C03632=1082.087,-21.908,442.728,174.022,19.619,153.310
C03633=1082.093,-21.658,442.716,174.024,19.621,153.310
C03634=1082.099,-21.409,442.702,174.025,19.623,153.310
C03635=1082.104,-21.158,442.689,174.026,19.625,153.311
C03636=1082.110,-20.909,442.676,174.028,19.627,153.311
C03637=1082.116,-20.659,442.663,174.030,19.629,153.311
C03638=1082.122,-20.410,442.650,174.031,19.631,153.311
C03639=1082.128,-20.160,442.636,174.032,19.633,153.311
C03640=1082.134,-19.910,442.624,174.034,19.635,153.311
C03641=1082.140,-19.661,442.610,174.035,19.637,153.311
C03642=1082.146,-19.411,442.598,174.037,19.639,153.311
C03643=1082.152,-19.162,442.585,174.039,19.641,153.312
C03644=1082.157,-18.912,442.571,174.040,19.643,153.312
C03645=1082.164,-18.663,442.558,174.041,19.645,153.312
C03646=1082.170,-18.413,442.545,174.042,19.647,153.312
C03647=1082.176,-18.163,442.532,174.045,19.649,153.312
C03648=1082.181,-17.914,442.518,174.046,19.651,153.312
C03649=1082.187,-17.664,442.506,174.047,19.653,153.312
C03650=1082.194,-17.391,442.491,174.048,19.655,153.313
C03651=1082.200,-17.116,442.477,174.050,19.658,153.313
C03652=1082.206,-16.843,442.462,174.052,19.660,153.313
C03653=1082.213,-16.568,442.448,174.054,19.662,153.313
C03654=1082.220,-16.319,442.435,174.055,19.664,153.313
C03655=1082.225,-16.069,442.421,174.056,19.666,153.313
C03656=1082.231,-15.819,442.408,174.058,19.668,153.313
C03657=1082.237,-15.570,442.395,174.059,19.670,153.314
C03658=1082.243,-15.321,442.382,174.061,19.672,153.314
C03659=1082.249,-15.071,442.369,174.063,19.674,153.314
C03660=1082.255,-14.821,442.355,174.064,19.676,153.314
C03661=1082.260,-14.572,442.341,174.065,19.678,153.314
C03662=1082.266,-14.322,442.329,174.066,19.680,153.314
C03663=1082.272,-14.073,442.316,174.068,19.682,153.314
C03664=1082.278,-13.823,442.302,174.070,19.684,153.314
C03665=1082.284,-13.574,442.288,174.071,19.686,153.315
C03666=1082.289,-13.324,442.275,174.072,19.688,153.315
C03667=1082.295,-13.074,442.262,174.074,19.690,153.315
C03668=1082.301,-12.825,442.248,174.076,19.692,153.315
C03669=1082.307,-12.576,442.235,174.077,19.694,153.315
C03670=1082.312,-12.325,442.222,174.078,19.696,153.315
C03671=1082.319,-12.076,442.208,174.079,19.698,153.316
C03672=1082.324,-11.827,442.195,174.082,19.700,153.316
C03673=1082.330,-11.577,442.181,174.083,19.702,153.316
C03674=1082.336,-11.328,442.167,174.084,19.704,153.316
C03675=1082.342,-11.078,442.155,174.085,19.706,153.316
C03676=1082.348,-10.828,442.141,174.087,19.708,153.316
C03677=1082.354,-10.578,442.127,174.089,19.711,153.316
C03678=1082.360,-10.329,442.114,174.090,19.713,153.317
C03679=1082.366,-10.079,442.100,174.091,19.714,153.317
C03680=1082.372,-9.830,442.087,174.093,19.716,153.317
C03681=1082.377,-9.580,442.074,174.095,19.719,153.317
C03682=1082.383,-9.331,442.061,174.096,19.721,153.317
C03683=1082.389,-9.081,442.047,174.097,19.723,153.317
C03684=1082.395,-8.832,442.033,174.099,19.725,153.318
C03685=1082.400,-8.582,442.020,174.100,19.727,153.318
C03686=1082.407,-8.333,442.006,174.102,19.729,153.318
C03687=1082.413,-8.083,441.992,174.103,19.731,153.318
C03688=1082.418,-7.833,441.978,174.105,19.733,153.318
C03689=1082.424,-7.584,441.965,174.106,19.735,153.318
C03690=1082.430,-7.334,441.952,174.108,19.738,153.318
C03691=1082.436,-7.084,441.939,174.109,19.740,153.319
C03692=1082.441,-6.835,441.925,174.110,19.742,153.319
C03693=1082.447,-6.586,441.911,174.112,19.743,153.319
C03694=1082.454,-6.335,441.897,174.113,19.745,153.319
C03695=1082.460,-6.086,441.884,174.115,19.748,153.319
C03696=1082.465,-5.837,441.870,174.117,19.750,153.319
C03697=1082.471,-5.587,441.857,174.118,19.752,153.319
C03698=1082.477,-5.338,441.843,174.119,19.754,153.320
C03699=1082.483,-5.088,441.830,174.121,19.756,153.320
C03700=1082.489,-4.839,441.816,174.123,19.758,153.320
C03701=1082.495,-4.589,441.802,174.124,19.760,153.320
C03702=1082.501,-4.339,441.788,174.125,19.762,153.320
C03703=1082.506,-4.090,441.774,174.127,19.764,153.320
C03704=1082.513,-3.840,441.761,174.128,19.766,153.320
C03705=1082.518,-3.591,441.747,174.130,19.768,153.321
C03706=1082.525,-3.341,441.734,174.131,19.770,153.321
C03707=1082.530,-3.091,441.720,174.132,19.772,153.321
C03708=1082.536,-2.842,441.706,174.134,19.775,153.321
C03709=1082.541,-2.592,441.692,174.136,19.776,153.321
C03710=1082.548,-2.343,441.679,174.137,19.778,153.321
C03711=1082.553,-2.094,441.664,174.138,19.780,153.321
C03712=1082.559,-1.844,441.650,174.140,19.783,153.322
C03713=1082.565,-1.594,441.636,174.142,19.785,153.322
C03714=1082.571,-1.319,441.621,174.143,19.787,153.322
C03715=1082.577,-1.043,441.605,174.145,19.790,153.322
C03716=1082.584,-0.768,441.591,174.146,19.792,153.322
C03717=1082.590,-0.492,441.575,174.148,19.794,153.322
C03718=1082.596,-0.243,441.561,174.149,19.796,153.323
C03719=1082.602,0.007,441.548,174.151,19.798,153.323
C03720=1082.607,0.256,441.534,174.153,19.801,153.323
C03721=1082.613,0.507,441.520,174.154,19.803,153.323
C03722=1082.619,0.756,441.506,174.155,19.805,153.323
C03723=1082.625,1.005,441.492,174.156,19.807,153.323
C03724=1082.631,1.255,441.478,174.158,19.809,153.324
C03725=1082.636,1.504,441.464,174.160,19.811,153.324
C03726=1082.642,1.754,441.450,174.161,19.813,153.324
C03727=1082.648,2.004,441.436,174.162,19.815,153.324
C03728=1082.653,2.253,441.421,174.164,19.818,153.324
C03729=1082.660,2.502,441.408,174.166,19.820,153.324
C03730=1082.665,2.752,441.394,174.167,19.821,153.324
C03731=1082.671,3.002,441.380,174.168,19.823,153.325
C03732=1082.677,3.252,441.366,174.170,19.826,153.325
C03733=1082.682,3.501,441.351,174.172,19.828,153.325
C03734=1082.688,3.750,441.338,174.173,19.830,153.325
C03735=1082.694,4.000,441.323,174.174,19.832,153.325
C03736=1082.701,4.249,441.309,174.176,19.834,153.325
C03737=1082.706,4.499,441.296,174.178,19.836,153.326
C03738=1082.711,4.748,441.282,174.179,19.838,153.326
C03739=1082.718,4.999,441.267,174.180,19.840,153.326
C03740=1082.723,5.247,441.253,174.182,19.843,153.326
C03741=1082.729,5.497,441.239,174.183,19.845,153.326
C03742=1082.734,5.747,441.225,174.185,19.847,153.326
C03743=1082.741,5.996,441.210,174.186,19.849,153.327
C03744=1082.747,6.246,441.197,174.188,19.851,153.327
C03745=1082.752,6.495,441.183,174.189,19.853,153.327
C03746=1082.759,6.745,441.168,174.190,19.855,153.327
C03747=1082.764,6.994,441.154,174.192,19.857,153.327
C03748=1082.770,7.244,441.140,174.194,19.859,153.327
C03749=1082.776,7.494,441.125,174.195,19.861,153.327
C03750=1082.782,7.743,441.112,174.197,19.863,153.328
C03751=1082.787,7.993,441.098,174.199,19.866,153.328
C03752=1082.793,8.242,441.083,174.200,19.868,153.328
C03753=1082.799,8.492,441.069,174.201,19.870,153.328
C03754=1082.805,8.741,441.055,174.202,19.872,153.328
C03755=1082.811,8.991,441.041,174.205,19.874,153.328
C03756=1082.817,9.240,441.026,174.206,19.876,153.329
C03757=1082.823,9.489,441.012,174.207,19.878,153.329
C03758=1082.829,9.740,440.998,174.208,19.880,153.329
C03759=1082.835,9.989,440.983,174.210,19.883,153.329
C03760=1082.840,10.238,440.970,174.212,19.884,153.329
C03761=1082.846,10.488,440.955,174.213,19.886,153.329
C03762=1082.852,10.737,440.941,174.214,19.888,153.330
C03763=1082.858,10.986,440.926,174.217,19.891,153.330
C03764=1082.864,11.237,440.912,174.218,19.893,153.330
C03765=1082.870,11.486,440.897,174.219,19.895,153.330
C03766=1082.876,11.736,440.883,174.221,19.897,153.330
C03767=1082.881,11.985,440.869,174.222,19.899,153.330
C03768=1082.887,12.234,440.855,174.224,19.902,153.330
C03769=1082.893,12.484,440.840,174.225,19.904,153.331
C03770=1082.899,12.734,440.826,174.227,19.906,153.331
C03771=1082.905,12.983,440.811,174.228,19.907,153.331
C03772=1082.911,13.233,440.797,174.230,19.909,153.331
C03773=1082.917,13.482,440.783,174.231,19.911,153.331
C03774=1082.924,13.731,440.768,174.233,19.914,153.331
C03775=1082.929,13.981,440.754,174.234,19.916,153.332
C03776=1082.935,14.230,440.739,174.236,19.918,153.332
C03777=1082.941,14.480,440.725,174.238,19.920,153.332
C03778=1082.947,14.757,440.709,174.239,19.922,153.332
C03779=1082.954,15.035,440.693,174.241,19.925,153.332
C03780=1082.960,15.313,440.677,174.242,19.927,153.332
C03781=1082.967,15.590,440.661,174.244,19.930,153.333
C03782=1082.972,15.840,440.646,174.245,19.932,153.333
C03783=1082.978,16.089,440.631,174.247,19.934,153.333
C03784=1082.984,16.339,440.616,174.249,19.936,153.333
C03785=1082.990,16.588,440.602,174.250,19.938,153.333
C03786=1082.995,16.837,440.588,174.252,19.940,153.333
C03787=1083.002,17.087,440.573,174.253,19.942,153.333
C03788=1083.006,17.337,440.558,174.255,19.944,153.334
C03789=1083.013,17.587,440.543,174.256,19.946,153.334
C03790=1083.019,17.836,440.529,174.257,19.948,153.334
C03791=1083.025,18.086,440.515,174.260,19.951,153.334
C03792=1083.030,18.335,440.500,174.261,19.953,153.334
C03793=1083.035,18.584,440.485,174.262,19.955,153.334
C03794=1083.042,18.834,440.471,174.263,19.957,153.335
C03795=1083.047,19.083,440.456,174.265,19.959,153.335
C03796=1083.054,19.333,440.441,174.267,19.961,153.335
C03797=1083.059,19.582,440.426,174.268,19.963,153.335
C03798=1083.065,19.833,440.412,174.270,19.966,153.335
C03799=1083.071,20.081,440.397,174.271,19.968,153.335
C03800=1083.077,20.331,440.382,174.273,19.970,153.336
C03801=1083.083,20.580,440.368,174.275,19.972,153.336
C03802=1083.088,20.831,440.353,174.276,19.974,153.336
C03803=1083.094,21.080,440.338,174.277,19.976,153.336
C03804=1083.100,21.329,440.324,174.278,19.978,153.336
C03805=1083.105,21.579,440.308,174.281,19.981,153.336
C03806=1083.111,21.828,440.293,174.282,19.983,153.337
C03807=1083.117,22.078,440.279,174.283,19.985,153.337
C03808=1083.123,22.327,440.265,174.285,19.987,153.337
C03809=1083.129,22.577,440.249,174.286,19.989,153.337
C03810=1083.134,22.826,440.235,174.288,19.991,153.337
C03811=1083.141,23.075,440.220,174.290,19.993,153.337
C03812=1083.146,23.325,440.204,174.291,19.995,153.337
C03813=1083.152,23.574,440.189,174.293,19.997,153.338
C03814=1083.158,23.824,440.176,174.294,19.999,153.338
C03815=1083.163,24.074,440.160,174.296,20.002,153.338
C03816=1083.169,24.323,440.145,174.297,20.004,153.338
C03817=1083.175,24.573,440.130,174.298,20.006,153.338
C03818=1083.181,24.822,440.115,174.301,20.008,153.338
C03819=1083.187,25.071,440.100,174.302,20.010,153.339
C03820=1083.192,25.321,440.085,174.303,20.012,153.339
C03821=1083.198,25.570,440.070,174.305,20.015,153.339
C03822=1083.204,25.819,440.056,174.306,20.017,153.339
C03823=1083.210,26.069,440.040,174.308,20.019,153.339
C03824=1083.216,26.319,440.025,174.310,20.021,153.339
C03825=1083.222,26.568,440.011,174.311,20.023,153.340
C03826=1083.227,26.818,439.996,174.312,20.025,153.340
C03827=1083.233,27.067,439.981,174.315,20.028,153.340
C03828=1083.239,27.317,439.966,174.316,20.030,153.340
C03829=1083.244,27.566,439.951,174.317,20.031,153.340
C03830=1083.251,27.816,439.936,174.319,20.033,153.340
C03831=1083.256,28.065,439.921,174.321,20.036,153.340
C03832=1083.262,28.315,439.906,174.322,20.038,153.341
C03833=1083.268,28.565,439.891,174.323,20.040,153.341
C03834=1083.274,28.813,439.875,174.325,20.042,153.341
C03835=1083.280,29.063,439.860,174.327,20.044,153.341
C03836=1083.285,29.312,439.845,174.328,20.046,153.341
C03837=1083.291,29.562,439.830,174.330,20.049,153.341
C03838=1083.297,29.811,439.815,174.331,20.051,153.342
C03839=1083.303,30.061,439.799,174.332,20.053,153.342
C03840=1083.308,30.310,439.785,174.335,20.055,153.342
C03841=1083.314,30.560,439.769,174.336,20.057,153.342
C03842=1083.321,30.839,439.753,174.338,20.060,153.342
C03843=1083.327,31.118,439.735,174.339,20.062,153.342
C03844=1083.333,31.397,439.719,174.341,20.065,153.343
C03845=1083.340,31.676,439.701,174.342,20.067,153.343
C03846=1083.345,31.925,439.687,174.344,20.069,153.343
C03847=1083.351,32.175,439.670,174.346,20.071,153.343
C03848=1083.357,32.424,439.656,174.347,20.073,153.343
C03849=1083.363,32.674,439.640,174.349,20.076,153.343
C03850=1083.368,32.924,439.625,174.351,20.077,153.343
C03851=1083.374,33.173,439.610,174.352,20.079,153.344
C03852=1083.380,33.422,439.595,174.354,20.082,153.344
C03853=1083.386,33.672,439.580,174.355,20.084,153.344
C03854=1083.392,33.921,439.564,174.357,20.086,153.344
C03855=1083.397,34.171,439.548,174.359,20.088,153.344
C03856=1083.403,34.420,439.534,174.360,20.090,153.344
C03857=1083.409,34.670,439.518,174.361,20.092,153.345
C03858=1083.415,34.919,439.502,174.363,20.095,153.345
C03859=1083.420,35.168,439.487,174.365,20.097,153.345
C03860=1083.426,35.418,439.472,174.366,20.099,153.345
C03861=1083.432,35.668,439.457,174.368,20.101,153.345
C03862=1083.437,35.917,439.442,174.369,20.103,153.345
C03863=1083.444,36.166,439.426,174.371,20.105,153.345
C03864=1083.450,36.416,439.410,174.373,20.107,153.346
C03865=1083.455,36.665,439.395,174.374,20.109,153.346
C03866=1083.462,36.914,439.380,174.375,20.111,153.346
C03867=1083.467,37.164,439.364,174.377,20.113,153.346
C03868=1083.472,37.413,439.349,174.379,20.115,153.346
C03869=1083.479,37.662,439.333,174.380,20.117,153.346
C03870=1083.485,37.912,439.318,174.382,20.120,153.347
C03871=1083.490,38.162,439.302,174.383,20.122,153.347
C03872=1083.496,38.411,439.288,174.385,20.124,153.347
C03873=1083.502,38.661,439.271,174.387,20.126,153.347
C03874=1083.508,38.911,439.256,174.388,20.128,153.347
C03875=1083.513,39.159,439.240,174.390,20.131,153.347
C03876=1083.519,39.409,439.224,174.392,20.132,153.347
C03877=1083.525,39.659,439.209,174.393,20.134,153.348
C03878=1083.530,39.908,439.194,174.395,20.137,153.348
C03879=1083.536,40.158,439.178,174.396,20.139,153.348
C03880=1083.542,40.408,439.162,174.398,20.141,153.348
C03881=1083.547,40.656,439.147,174.400,20.143,153.348
C03882=1083.553,40.906,439.132,174.401,20.145,153.348
C03883=1083.559,41.155,439.115,174.402,20.147,153.349
C03884=1083.564,41.404,439.100,174.404,20.150,153.349
C03885=1083.570,41.654,439.084,174.406,20.152,153.349
C03886=1083.576,41.904,439.068,174.407,20.154,153.349
C03887=1083.582,42.153,439.053,174.409,20.156,153.349
C03888=1083.588,42.402,439.038,174.410,20.158,153.349
C03889=1083.593,42.652,439.022,174.412,20.161,153.350
C03890=1083.599,42.901,439.006,174.414,20.162,153.350
C03891=1083.605,43.151,438.990,174.415,20.164,153.350
C03892=1083.610,43.400,438.974,174.417,20.167,153.350
C03893=1083.617,43.650,438.959,174.419,20.169,153.350
C03894=1083.623,43.899,438.943,174.420,20.171,153.350
C03895=1083.628,44.149,438.928,174.422,20.173,153.350
C03896=1083.634,44.398,438.912,174.423,20.175,153.351
C03897=1083.639,44.648,438.896,174.424,20.177,153.351
C03898=1083.645,44.897,438.880,174.427,20.180,153.351
C03899=1083.650,45.146,438.865,174.428,20.182,153.351
C03900=1083.656,45.396,438.848,174.430,20.184,153.351
C03901=1083.662,45.645,438.832,174.431,20.186,153.351
C03902=1083.668,45.895,438.817,174.433,20.188,153.352
C03903=1083.673,46.144,438.801,174.435,20.190,153.352
C03904=1083.678,46.394,438.785,174.436,20.192,153.352
C03905=1083.684,46.643,438.768,174.437,20.194,153.352
C03906=1083.690,46.923,438.751,174.439,20.197,153.352
C03907=1083.697,47.201,438.733,174.441,20.199,153.352
C03908=1083.703,47.480,438.715,174.443,20.201,153.353
C03909=1083.709,47.759,438.698,174.445,20.204,153.353
C03910=1083.715,48.008,438.681,174.446,20.206,153.353
C03911=1083.721,48.258,438.665,174.448,20.208,153.353
C03912=1083.726,48.508,438.650,174.450,20.210,153.353
C03913=1083.732,48.756,438.634,174.452,20.213,153.353
C03914=1083.738,49.006,438.618,174.453,20.215,153.353
C03915=1083.743,49.256,438.602,174.454,20.217,153.354
C03916=1083.749,49.505,438.586,174.456,20.219,153.354
C03917=1083.755,49.754,438.569,174.458,20.221,153.354
C03918=1083.760,50.004,438.554,174.460,20.224,153.354
C03919=1083.766,50.253,438.538,174.461,20.225,153.354
C03920=1083.772,50.502,438.522,174.462,20.227,153.354
C03921=1083.778,50.752,438.506,174.465,20.230,153.354
C03922=1083.783,51.002,438.489,174.466,20.232,153.355
C03923=1083.789,51.251,438.473,174.467,20.234,153.355
C03924=1083.794,51.500,438.457,174.469,20.236,153.355
C03925=1083.800,51.749,438.441,174.471,20.238,153.355
C03926=1083.806,51.999,438.425,174.473,20.240,153.355
C03927=1083.812,52.249,438.409,174.474,20.242,153.355
C03928=1083.818,52.498,438.393,174.475,20.244,153.356
C03929=1083.824,52.747,438.377,174.478,20.246,153.356
C03930=1083.829,52.997,438.361,174.479,20.248,153.356
C03931=1083.834,53.246,438.345,174.481,20.251,153.356
C03932=1083.840,53.496,438.328,174.482,20.253,153.356
C03933=1083.846,53.745,438.312,174.484,20.255,153.356
C03934=1083.852,53.994,438.296,174.486,20.257,153.356
C03935=1083.858,54.244,438.280,174.487,20.259,153.356
C03936=1083.863,54.494,438.264,174.489,20.261,153.357
C03937=1083.869,54.743,438.248,174.491,20.263,153.357
C03938=1083.875,54.992,438.232,174.492,20.265,153.357
C03939=1083.880,55.241,438.215,174.494,20.268,153.357
C03940=1083.886,55.491,438.199,174.495,20.269,153.357
C03941=1083.892,55.740,438.183,174.498,20.272,153.357
C03942=1083.898,55.989,438.166,174.499,20.274,153.357
C03943=1083.904,56.239,438.150,174.500,20.276,153.358
C03944=1083.910,56.488,438.134,174.502,20.278,153.358
C03945=1083.915,56.738,438.118,174.504,20.280,153.358
C03946=1083.921,56.988,438.101,174.506,20.282,153.358
C03947=1083.927,57.237,438.085,174.507,20.284,153.358
C03948=1083.932,57.486,438.069,174.508,20.286,153.358
C03949=1083.938,57.736,438.053,174.511,20.288,153.358
C03950=1083.944,57.985,438.036,174.512,20.290,153.359
C03951=1083.950,58.235,438.020,174.514,20.292,153.359
C03952=1083.956,58.484,438.003,174.516,20.294,153.359
C03953=1083.962,58.733,437.987,174.517,20.296,153.359
C03954=1083.967,58.983,437.971,174.519,20.298,153.359
C03955=1083.973,59.232,437.954,174.520,20.300,153.359
C03956=1083.979,59.482,437.938,174.523,20.303,153.359
C03957=1083.985,59.731,437.921,174.524,20.305,153.360
C03958=1083.991,59.980,437.905,174.525,20.306,153.360
C03959=1083.996,60.230,437.889,174.527,20.309,153.360
C03960=1084.002,60.479,437.872,174.529,20.311,153.360
C03961=1084.008,60.729,437.856,174.531,20.313,153.360
C03962=1084.014,60.977,437.839,174.532,20.315,153.360
C03963=1084.020,61.227,437.823,174.534,20.317,153.360
C03964=1084.026,61.476,437.806,174.536,20.319,153.360
C03965=1084.031,61.726,437.789,174.537,20.321,153.360
C03966=1084.037,61.975,437.773,174.539,20.323,153.361
C03967=1084.043,62.225,437.757,174.541,20.325,153.361
C03968=1084.049,62.474,437.741,174.543,20.327,153.361
C03969=1084.054,62.724,437.724,174.544,20.329,153.361
C03970=1084.061,63.002,437.705,174.546,20.331,153.361
C03971=1084.067,63.281,437.687,174.548,20.333,153.361
C03972=1084.074,63.559,437.669,174.550,20.336,153.361
C03973=1084.080,63.838,437.651,174.552,20.338,153.362
C03974=1084.087,64.088,437.633,174.554,20.340,153.362
C03975=1084.093,64.337,437.616,174.556,20.342,153.362
C03976=1084.098,64.587,437.600,174.557,20.344,153.362
C03977=1084.104,64.836,437.583,174.558,20.346,153.362
C03978=1084.110,65.086,437.567,174.561,20.348,153.362
C03979=1084.115,65.335,437.550,174.562,20.350,153.362
C03980=1084.121,65.584,437.533,174.564,20.353,153.362
C03981=1084.127,65.833,437.517,174.565,20.354,153.362
C03982=1084.132,66.083,437.500,174.568,20.356,153.363
C03983=1084.139,66.332,437.483,174.569,20.358,153.363
C03984=1084.144,66.581,437.466,174.571,20.361,153.363
C03985=1084.150,66.831,437.450,174.573,20.362,153.363
C03986=1084.155,67.080,437.433,174.574,20.364,153.363
C03987=1084.161,67.329,437.416,174.576,20.367,153.363
C03988=1084.166,67.579,437.399,174.577,20.369,153.363
C03989=1084.172,67.828,437.383,174.580,20.371,153.363
C03990=1084.178,68.078,437.366,174.581,20.373,153.364
C03991=1084.184,68.327,437.349,174.583,20.375,153.364
C03992=1084.190,68.577,437.332,174.585,20.377,153.364
C03993=1084.196,68.826,437.316,174.586,20.379,153.364
C03994=1084.201,69.075,437.298,174.588,20.381,153.364
C03995=1084.207,69.325,437.282,174.589,20.383,153.364
C03996=1084.212,69.574,437.265,174.592,20.385,153.364
C03997=1084.218,69.823,437.248,174.593,20.387,153.364
C03998=1084.224,70.073,437.231,174.595,20.389,153.365
C03999=1084.229,70.322,437.214,174.596,20.391,153.365
C04000=1084.235,70.571,437.198,174.599,20.393,153.365
C04001=1084.240,70.821,437.181,174.600,20.395,153.365
C04002=1084.247,71.070,437.163,174.601,20.397,153.365
C04003=1084.252,71.320,437.146,174.604,20.399,153.365
C04004=1084.258,71.569,437.129,174.605,20.401,153.365
C04005=1084.264,71.818,437.113,174.607,20.404,153.365
C04006=1084.269,72.068,437.096,174.608,20.405,153.366
C04007=1084.275,72.317,437.078,174.611,20.408,153.366
C04008=1084.281,72.566,437.062,174.612,20.410,153.366
C04009=1084.286,72.815,437.044,174.614,20.412,153.366
C04010=1084.291,73.065,437.028,174.616,20.414,153.366
C04011=1084.298,73.314,437.010,174.618,20.416,153.366
C04012=1084.303,73.564,436.993,174.619,20.417,153.366
C04013=1084.309,73.813,436.976,174.620,20.419,153.366
C04014=1084.315,74.063,436.960,174.623,20.422,153.367
C04015=1084.320,74.312,436.942,174.624,20.423,153.367
C04016=1084.326,74.561,436.925,174.626,20.426,153.367
C04017=1084.332,74.811,436.908,174.628,20.428,153.367
C04018=1084.338,75.060,436.891,174.630,20.430,153.367
C04019=1084.343,75.309,436.873,174.631,20.432,153.367
C04020=1084.349,75.559,436.857,174.633,20.434,153.367
C04021=1084.355,75.808,436.840,174.635,20.436,153.367
C04022=1084.360,76.057,436.822,174.637,20.438,153.367
C04023=1084.367,76.307,436.805,174.638,20.440,153.368
C04024=1084.372,76.556,436.788,174.641,20.442,153.368
C04025=1084.377,76.806,436.771,174.642,20.444,153.368
C04026=1084.383,77.055,436.753,174.643,20.445,153.368
C04027=1084.389,77.303,436.736,174.646,20.448,153.368
C04028=1084.395,77.554,436.719,174.647,20.450,153.368
C04029=1084.401,77.803,436.702,174.649,20.452,153.368
C04030=1084.406,78.052,436.685,174.650,20.454,153.368
C04031=1084.412,78.301,436.668,174.653,20.456,153.368
C04032=1084.418,78.550,436.650,174.654,20.458,153.368
C04033=1084.423,78.800,436.633,174.656,20.460,153.369
C04034=1084.429,79.079,436.614,174.658,20.463,153.369
C04035=1084.436,79.358,436.594,174.660,20.464,153.369
C04036=1084.442,79.636,436.575,174.662,20.467,153.369
C04037=1084.448,79.915,436.555,174.664,20.469,153.369
C04038=1084.455,80.164,436.538,174.665,20.471,153.369
C04039=1084.460,80.413,436.520,174.668,20.473,153.369
C04040=1084.465,80.663,436.504,174.669,20.475,153.369
C04041=1084.471,80.912,436.486,174.671,20.477,153.370
C04042=1084.477,81.161,436.468,174.673,20.479,153.370
C04043=1084.482,81.411,436.451,174.675,20.481,153.370
C04044=1084.488,81.660,436.434,174.676,20.483,153.370
C04045=1084.493,81.909,436.416,174.679,20.485,153.370
C04046=1084.499,82.159,436.398,174.680,20.487,153.370
C04047=1084.505,82.408,436.381,174.682,20.489,153.370
C04048=1084.510,82.658,436.364,174.684,20.491,153.370
C04049=1084.516,82.907,436.346,174.686,20.493,153.370
C04050=1084.522,83.156,436.328,174.687,20.495,153.371
C04051=1084.527,83.405,436.311,174.689,20.497,153.371
C04052=1084.533,83.654,436.294,174.691,20.499,153.371
C04053=1084.539,83.904,436.277,174.693,20.501,153.371
C04054=1084.545,84.154,436.259,174.694,20.503,153.371
C04055=1084.550,84.403,436.241,174.697,20.505,153.371
C04056=1084.556,84.652,436.224,174.698,20.507,153.371
C04057=1084.562,84.901,436.206,174.700,20.509,153.371
C04058=1084.567,85.150,436.188,174.702,20.511,153.371
C04059=1084.573,85.400,436.171,174.704,20.513,153.371
C04060=1084.579,85.649,436.153,174.705,20.515,153.372
C04061=1084.585,85.898,436.135,174.708,20.517,153.372
C04062=1084.590,86.148,436.118,174.709,20.519,153.372
C04063=1084.596,86.398,436.100,174.711,20.521,153.372
C04064=1084.601,86.647,436.083,174.713,20.523,153.372
C04065=1084.607,86.896,436.065,174.715,20.525,153.372
C04066=1084.613,87.146,436.047,174.716,20.527,153.372
C04067=1084.619,87.395,436.030,174.719,20.529,153.372
C04068=1084.624,87.644,436.012,174.720,20.531,153.372
C04069=1084.630,87.893,435.994,174.722,20.533,153.372
C04070=1084.636,88.142,435.977,174.724,20.535,153.373
C04071=1084.641,88.391,435.959,174.726,20.537,153.373
C04072=1084.647,88.641,435.941,174.727,20.538,153.373
C04073=1084.653,88.890,435.924,174.730,20.540,153.373
C04074=1084.658,89.139,435.906,174.731,20.542,153.373
C04075=1084.665,89.389,435.888,174.733,20.544,153.373
C04076=1084.670,89.638,435.871,174.735,20.546,153.373
C04077=1084.676,89.888,435.853,174.737,20.548,153.373
C04078=1084.681,90.137,435.835,174.738,20.550,153.373
C04079=1084.686,90.386,435.817,174.741,20.552,153.373
C04080=1084.693,90.636,435.799,174.742,20.554,153.373
C04081=1084.698,90.884,435.781,174.744,20.556,153.373
C04082=1084.705,91.134,435.763,174.746,20.558,153.373
C04083=1084.710,91.383,435.745,174.748,20.560,153.374
C04084=1084.716,91.632,435.728,174.749,20.561,153.374
C04085=1084.721,91.882,435.709,174.751,20.564,153.374
C04086=1084.727,92.131,435.692,174.753,20.565,153.374
C04087=1084.732,92.380,435.674,174.755,20.568,153.374
C04088=1084.738,92.630,435.656,174.757,20.569,153.374
C04089=1084.744,92.879,435.638,174.759,20.572,153.374
C04090=1084.749,93.128,435.619,174.760,20.573,153.374
C04091=1084.755,93.378,435.602,174.762,20.576,153.374
C04092=1084.760,93.627,435.584,174.765,20.577,153.374
C04093=1084.767,93.876,435.566,174.766,20.579,153.375
C04094=1084.771,94.126,435.548,174.768,20.581,153.375
C04095=1084.778,94.375,435.529,174.770,20.583,153.375
C04096=1084.783,94.624,435.512,174.772,20.585,153.375
C04097=1084.788,94.873,435.494,174.774,20.587,153.375
C04098=1084.795,95.152,435.474,174.776,20.589,153.375
C04099=1084.802,95.431,435.453,174.778,20.592,153.375
C04100=1084.807,95.710,435.433,174.780,20.594,153.375
C04101=1084.814,95.988,435.413,174.782,20.596,153.375
C04102=1084.820,96.237,435.395,174.784,20.597,153.375
C04103=1084.825,96.488,435.377,174.786,20.600,153.375
C04104=1084.831,96.736,435.358,174.788,20.601,153.375
C04105=1084.837,96.986,435.341,174.790,20.603,153.375
C04106=1084.842,97.235,435.323,174.791,20.605,153.376
C04107=1084.848,97.484,435.304,174.794,20.607,153.376
C04108=1084.854,97.733,435.286,174.795,20.609,153.376
C04109=1084.860,97.983,435.268,174.797,20.611,153.376
C04110=1084.865,98.232,435.249,174.799,20.613,153.376
C04111=1084.871,98.481,435.231,174.801,20.615,153.376
C04112=1084.876,98.730,435.214,174.803,20.616,153.376
C04113=1084.882,98.980,435.195,174.805,20.618,153.376
C04114=1084.888,99.229,435.177,174.807,20.621,153.376
C04115=1084.894,99.478,435.158,174.809,20.622,153.376
C04116=1084.899,99.727,435.140,174.811,20.624,153.376
C04117=1084.905,99.977,435.122,174.812,20.626,153.376
C04118=1084.911,100.226,435.104,174.815,20.628,153.376
C04119=1084.916,100.476,435.085,174.816,20.630,153.377
C04120=1084.922,100.724,435.067,174.818,20.632,153.377
C04121=1084.928,100.974,435.049,174.820,20.633,153.377
C04122=1084.933,101.223,435.031,174.822,20.635,153.377
C04123=1084.939,101.472,435.012,174.824,20.638,153.377
C04124=1084.944,101.722,434.994,174.826,20.639,153.377
C04125=1084.951,101.971,434.976,174.828,20.641,153.377
C04126=1084.955,102.220,434.957,174.830,20.643,153.377
C04127=1084.962,102.469,434.939,174.832,20.645,153.377
C04128=1084.967,102.719,434.921,174.833,20.647,153.377
C04129=1084.973,102.968,434.902,174.836,20.649,153.377
C04130=1084.978,103.218,434.883,174.838,20.651,153.377
C04131=1084.984,103.466,434.865,174.839,20.652,153.377
C04132=1084.990,103.716,434.847,174.842,20.655,153.377
C04133=1084.995,103.965,434.828,174.843,20.656,153.378
C04134=1085.001,104.214,434.809,174.845,20.659,153.378
C04135=1085.006,104.463,434.791,174.847,20.660,153.378
C04136=1085.012,104.713,434.772,174.849,20.662,153.378
C04137=1085.017,104.962,434.754,174.852,20.664,153.378
C04138=1085.023,105.211,434.736,174.853,20.666,153.378
C04139=1085.029,105.461,434.717,174.855,20.668,153.378
C04140=1085.034,105.710,434.698,174.857,20.669,153.378
C04141=1085.040,105.959,434.679,174.859,20.672,153.378
C04142=1085.045,106.208,434.661,174.860,20.673,153.378
C04143=1085.052,106.457,434.643,174.863,20.675,153.378
C04144=1085.057,106.706,434.624,174.865,20.678,153.378
C04145=1085.063,106.956,434.606,174.866,20.679,153.378
C04146=1085.068,107.205,434.587,174.869,20.681,153.378
C04147=1085.074,107.454,434.568,174.870,20.682,153.378
C04148=1085.080,107.704,434.550,174.872,20.685,153.379
C04149=1085.085,107.953,434.531,174.874,20.686,153.379
C04150=1085.091,108.202,434.512,174.876,20.688,153.379
C04151=1085.097,108.452,434.494,174.879,20.690,153.379
C04152=1085.102,108.700,434.475,174.880,20.692,153.379
C04153=1085.108,108.950,434.456,174.882,20.694,153.379
C04154=1085.113,109.200,434.438,174.884,20.696,153.379
C04155=1085.119,109.448,434.419,174.886,20.698,153.379
C04156=1085.125,109.697,434.400,174.889,20.699,153.379
C04157=1085.131,109.947,434.381,174.890,20.701,153.379
C04158=1085.136,110.195,434.363,174.892,20.703,153.379
C04159=1085.142,110.445,434.344,174.894,20.705,153.379
C04160=1085.148,110.695,434.325,174.896,20.707,153.379
C04161=1085.153,110.943,434.307,174.899,20.709,153.379
C04162=1085.160,111.222,434.285,174.900,20.711,153.379
C04163=1085.166,111.501,434.264,174.902,20.713,153.379
C04164=1085.172,111.780,434.243,174.905,20.714,153.379
C04165=1085.178,112.059,434.222,174.907,20.717,153.379
C04166=1085.184,112.308,434.203,174.909,20.719,153.379
C04167=1085.190,112.557,434.184,174.911,20.720,153.379
C04168=1085.196,112.806,434.165,174.913,20.722,153.379
C04169=1085.201,113.056,434.146,174.915,20.724,153.380
C04170=1085.207,113.306,434.128,174.917,20.726,153.380
C04171=1085.212,113.554,434.109,174.919,20.728,153.380
C04172=1085.218,113.803,434.090,174.921,20.729,153.380
C04173=1085.224,114.053,434.071,174.923,20.731,153.380
C04174=1085.229,114.302,434.052,174.925,20.733,153.380
C04175=1085.235,114.551,434.033,174.927,20.735,153.380
C04176=1085.241,114.800,434.014,174.929,20.737,153.380
C04177=1085.247,115.050,433.995,174.931,20.739,153.380
C04178=1085.252,115.298,433.976,174.933,20.741,153.380
C04179=1085.257,115.548,433.957,174.935,20.742,153.380
C04180=1085.263,115.797,433.938,174.937,20.744,153.380
C04181=1085.268,116.046,433.919,174.939,20.746,153.380
C04182=1085.274,116.295,433.899,174.941,20.748,153.380
C04183=1085.280,116.545,433.880,174.943,20.750,153.380
C04184=1085.285,116.794,433.861,174.945,20.752,153.380
C04185=1085.290,117.043,433.842,174.947,20.754,153.380
C04186=1085.296,117.292,433.823,174.949,20.756,153.380
C04187=1085.302,117.542,433.804,174.951,20.757,153.380
C04188=1085.307,117.791,433.785,174.953,20.759,153.381
C04189=1085.313,118.040,433.765,174.955,20.761,153.381
C04190=1085.318,118.289,433.746,174.957,20.763,153.381
C04191=1085.323,118.538,433.727,174.959,20.765,153.381
C04192=1085.329,118.788,433.708,174.961,20.767,153.381
C04193=1085.335,119.037,433.689,174.964,20.769,153.381
C04194=1085.340,119.286,433.670,174.965,20.770,153.381
C04195=1085.345,119.535,433.651,174.968,20.772,153.381
C04196=1085.351,119.784,433.631,174.970,20.774,153.381
C04197=1085.357,120.033,433.611,174.971,20.776,153.381
C04198=1085.363,120.283,433.592,174.974,20.778,153.381
C04199=1085.368,120.532,433.573,174.975,20.779,153.381
C04200=1085.374,120.781,433.554,174.978,20.781,153.381
C04201=1085.379,121.030,433.535,174.980,20.783,153.381
C04202=1085.385,121.280,433.516,174.981,20.784,153.381
C04203=1085.391,121.529,433.496,174.984,20.786,153.381
C04204=1085.396,121.777,433.477,174.986,20.788,153.381
C04205=1085.402,122.027,433.458,174.988,20.790,153.381
C04206=1085.407,122.276,433.438,174.990,20.792,153.381
C04207=1085.413,122.525,433.418,174.992,20.794,153.381
C04208=1085.419,122.775,433.399,174.994,20.796,153.381
C04209=1085.424,123.024,433.379,174.996,20.797,153.381
C04210=1085.429,123.273,433.360,174.999,20.799,153.381
C04211=1085.435,123.522,433.340,175.000,20.801,153.381
C04212=1085.441,123.771,433.321,175.002,20.803,153.381
C04213=1085.447,124.021,433.302,175.005,20.805,153.381
C04214=1085.452,124.270,433.283,175.006,20.806,153.382
C04215=1085.458,124.519,433.263,175.009,20.808,153.382
C04216=1085.464,124.768,433.244,175.011,20.810,153.382
C04217=1085.469,125.017,433.225,175.013,20.811,153.382
C04218=1085.475,125.266,433.205,175.015,20.813,153.382
C04219=1085.481,125.515,433.185,175.017,20.815,153.382
C04220=1085.486,125.765,433.166,175.019,20.817,153.382
C04221=1085.492,126.014,433.146,175.021,20.819,153.382
C04222=1085.497,126.263,433.126,175.024,20.821,153.382
C04223=1085.503,126.513,433.107,175.025,20.822,153.382
C04224=1085.509,126.762,433.087,175.028,20.824,153.382
C04225=1085.515,127.011,433.068,175.030,20.826,153.382
C04226=1085.521,127.289,433.046,175.032,20.828,153.382
C04227=1085.527,127.568,433.024,175.034,20.829,153.382
C04228=1085.533,127.847,433.003,175.036,20.831,153.382
C04229=1085.540,128.126,432.980,175.039,20.833,153.382
C04230=1085.545,128.376,432.961,175.041,20.835,153.382
C04231=1085.551,128.624,432.941,175.043,20.837,153.382
C04232=1085.557,128.874,432.921,175.046,20.839,153.382
C04233=1085.563,129.123,432.901,175.047,20.840,153.382
C04234=1085.568,129.371,432.883,175.050,20.842,153.382
C04235=1085.574,129.620,432.863,175.052,20.844,153.382
C04236=1085.579,129.870,432.843,175.054,20.845,153.382
C04237=1085.585,130.119,432.823,175.056,20.847,153.382
C04238=1085.591,130.368,432.804,175.059,20.849,153.382
C04239=1085.597,130.617,432.784,175.060,20.850,153.382
C04240=1085.602,130.866,432.764,175.062,20.852,153.382
C04241=1085.608,131.115,432.744,175.065,20.854,153.382
C04242=1085.614,131.364,432.724,175.067,20.855,153.382
C04243=1085.619,131.614,432.705,175.069,20.857,153.382
C04244=1085.625,131.863,432.685,175.071,20.859,153.382
C04245=1085.631,132.112,432.665,175.073,20.860,153.382
C04246=1085.636,132.361,432.645,175.075,20.862,153.382
C04247=1085.642,132.611,432.626,175.078,20.864,153.382
C04248=1085.648,132.859,432.606,175.080,20.866,153.382
C04249=1085.653,133.109,432.585,175.082,20.868,153.382
C04250=1085.659,133.358,432.566,175.084,20.870,153.382
C04251=1085.665,133.607,432.546,175.087,20.871,153.382
C04252=1085.670,133.856,432.525,175.088,20.872,153.382
C04253=1085.676,134.105,432.506,175.090,20.874,153.382
C04254=1085.681,134.354,432.486,175.093,20.876,153.382
C04255=1085.687,134.603,432.466,175.094,20.878,153.382
C04256=1085.693,134.853,432.446,175.097,20.880,153.382
C04257=1085.698,135.102,432.426,175.099,20.881,153.382
C04258=1085.704,135.351,432.406,175.101,20.883,153.382
C04259=1085.709,135.600,432.386,175.103,20.885,153.382
C04260=1085.715,135.849,432.366,175.106,20.886,153.382
C04261=1085.720,136.098,432.345,175.108,20.888,153.382
C04262=1085.726,136.347,432.326,175.110,20.890,153.382
C04263=1085.732,136.597,432.306,175.112,20.892,153.382
C04264=1085.738,136.846,432.285,175.114,20.893,153.382
C04265=1085.744,137.095,432.265,175.117,20.895,153.382
C04266=1085.749,137.344,432.245,175.118,20.897,153.382
C04267=1085.755,137.593,432.225,175.121,20.898,153.382
C04268=1085.760,137.843,432.205,175.123,20.900,153.382
C04269=1085.766,138.092,432.185,175.126,20.902,153.382
C04270=1085.771,138.341,432.165,175.127,20.903,153.382
C04271=1085.777,138.590,432.145,175.129,20.905,153.382
C04272=1085.783,138.839,432.124,175.132,20.907,153.382
C04273=1085.789,139.088,432.104,175.134,20.908,153.382
C04274=1085.793,139.337,432.084,175.136,20.910,153.382
C04275=1085.799,139.586,432.064,175.138,20.912,153.382
C04276=1085.805,139.835,432.044,175.141,20.914,153.382
C04277=1085.811,140.085,432.023,175.142,20.915,153.382
C04278=1085.817,140.334,432.003,175.145,20.917,153.382
C04279=1085.823,140.583,431.983,175.147,20.919,153.382
C04280=1085.828,140.832,431.962,175.150,20.921,153.382
C04281=1085.833,141.081,431.942,175.151,20.922,153.382
C04282=1085.839,141.330,431.922,175.154,20.924,153.382
C04283=1085.844,141.579,431.901,175.156,20.925,153.382
C04284=1085.850,141.828,431.881,175.159,20.927,153.382
C04285=1085.856,142.077,431.861,175.160,20.929,153.382
C04286=1085.861,142.327,431.841,175.162,20.931,153.382
C04287=1085.866,142.576,431.820,175.165,20.933,153.382
C04288=1085.872,142.825,431.800,175.167,20.934,153.382
C04289=1085.878,143.074,431.779,175.169,20.936,153.382
C04290=1085.884,143.352,431.756,175.171,20.937,153.382
C04291=1085.890,143.632,431.734,175.175,20.940,153.382
C04292=1085.896,143.910,431.710,175.177,20.942,153.382
C04293=1085.903,144.189,431.688,175.179,20.944,153.382
C04294=1085.909,144.438,431.668,175.182,20.945,153.382
C04295=1085.914,144.687,431.647,175.183,20.946,153.382
C04296=1085.919,144.936,431.627,175.186,20.948,153.382
C04297=1085.924,145.185,431.606,175.188,20.950,153.382
C04298=1085.931,145.433,431.585,175.191,20.952,153.382
C04299=1085.937,145.683,431.564,175.192,20.953,153.382
C04300=1085.942,145.932,431.544,175.195,20.955,153.382
C04301=1085.948,146.181,431.524,175.197,20.956,153.382
C04302=1085.953,146.430,431.503,175.200,20.958,153.382
C04303=1085.958,146.679,431.483,175.201,20.960,153.382
C04304=1085.965,146.929,431.463,175.204,20.961,153.382
C04305=1085.971,147.177,431.441,175.206,20.963,153.382
C04306=1085.976,147.426,431.421,175.209,20.965,153.382
C04307=1085.981,147.676,431.400,175.211,20.966,153.381
C04308=1085.988,147.925,431.380,175.213,20.968,153.382
C04309=1085.993,148.174,431.359,175.215,20.970,153.382
C04310=1085.998,148.423,431.338,175.218,20.971,153.381
C04311=1086.004,148.672,431.317,175.220,20.973,153.381
C04312=1086.009,148.921,431.297,175.222,20.975,153.381
C04313=1086.015,149.171,431.276,175.224,20.977,153.381
C04314=1086.021,149.419,431.255,175.227,20.978,153.381
C04315=1086.026,149.668,431.235,175.229,20.980,153.381
C04316=1086.032,149.917,431.214,175.231,20.982,153.381
C04317=1086.037,150.167,431.193,175.233,20.983,153.381
C04318=1086.043,150.416,431.172,175.236,20.985,153.381
C04319=1086.048,150.665,431.151,175.238,20.987,153.381
C04320=1086.054,150.914,431.131,175.241,20.988,153.381
C04321=1086.060,151.163,431.109,175.243,20.990,153.381
C04322=1086.066,151.412,431.089,175.244,20.991,153.381
C04323=1086.071,151.661,431.069,175.247,20.993,153.381
C04324=1086.077,151.909,431.047,175.249,20.995,153.381
C04325=1086.082,152.159,431.027,175.252,20.996,153.381
C04326=1086.088,152.408,431.006,175.254,20.998,153.381
C04327=1086.093,152.657,430.985,175.256,20.999,153.381
C04328=1086.098,152.906,430.964,175.258,21.001,153.381
C04329=1086.105,153.155,430.943,175.261,21.003,153.381
C04330=1086.110,153.404,430.922,175.263,21.005,153.381
C04331=1086.115,153.654,430.901,175.266,21.006,153.381
C04332=1086.121,153.903,430.880,175.267,21.007,153.381
C04333=1086.127,154.152,430.859,175.270,21.009,153.381
C04334=1086.132,154.400,430.838,175.272,21.011,153.381
C04335=1086.138,154.650,430.817,175.275,21.013,153.381
C04336=1086.144,154.899,430.796,175.277,21.015,153.381
C04337=1086.149,155.148,430.775,175.280,21.016,153.381
C04338=1086.155,155.397,430.754,175.281,21.017,153.381
C04339=1086.160,155.646,430.733,175.284,21.019,153.381
C04340=1086.166,155.895,430.712,175.286,21.021,153.381
C04341=1086.172,156.144,430.691,175.289,21.023,153.381
C04342=1086.177,156.393,430.670,175.291,21.024,153.381
C04343=1086.182,156.642,430.649,175.294,21.026,153.381
C04344=1086.189,156.891,430.627,175.295,21.027,153.381
C04345=1086.194,157.140,430.607,175.298,21.029,153.381
C04346=1086.199,157.389,430.586,175.300,21.031,153.381
C04347=1086.206,157.638,430.564,175.303,21.032,153.380
C04348=1086.210,157.888,430.543,175.305,21.034,153.380
C04349=1086.216,158.136,430.522,175.308,21.035,153.380
C04350=1086.222,158.386,430.501,175.309,21.037,153.380
C04351=1086.227,158.634,430.479,175.312,21.038,153.380
C04352=1086.233,158.884,430.458,175.314,21.040,153.380
C04353=1086.239,159.133,430.437,175.317,21.042,153.380
C04354=1086.245,159.411,430.412,175.319,21.044,153.380
C04355=1086.251,159.689,430.389,175.322,21.045,153.380
C04356=1086.258,159.968,430.366,175.325,21.047,153.380
C04357=1086.264,160.247,430.342,175.328,21.049,153.380
C04358=1086.269,160.495,430.320,175.330,21.051,153.380
C04359=1086.275,160.744,430.299,175.332,21.052,153.380
C04360=1086.281,160.994,430.278,175.334,21.053,153.380
C04361=1086.286,161.242,430.257,175.337,21.055,153.380
C04362=1086.292,161.492,430.235,175.339,21.057,153.380
C04363=1086.297,161.740,430.213,175.342,21.059,153.380
C04364=1086.302,161.989,430.193,175.344,21.061,153.380
C04365=1086.308,162.239,430.171,175.347,21.062,153.380
C04366=1086.313,162.487,430.149,175.348,21.063,153.380
C04367=1086.318,162.736,430.127,175.351,21.065,153.380
C04368=1086.324,162.985,430.106,175.353,21.067,153.380
C04369=1086.330,163.234,430.085,175.356,21.069,153.380
C04370=1086.335,163.484,430.063,175.358,21.071,153.380
C04371=1086.341,163.732,430.042,175.361,21.072,153.379
C04372=1086.345,163.981,430.020,175.363,21.074,153.380
C04373=1086.352,164.230,429.998,175.366,21.075,153.379
C04374=1086.357,164.479,429.977,175.367,21.077,153.379
C04375=1086.362,164.729,429.956,175.370,21.079,153.379
C04376=1086.368,164.978,429.934,175.372,21.080,153.379
C04377=1086.373,165.226,429.912,175.375,21.082,153.379
C04378=1086.379,165.476,429.891,175.377,21.083,153.379
C04379=1086.384,165.724,429.869,175.380,21.085,153.379
C04380=1086.390,165.974,429.847,175.382,21.087,153.379
C04381=1086.395,166.222,429.825,175.385,21.089,153.379
C04382=1086.401,166.472,429.804,175.387,21.090,153.379
C04383=1086.406,166.720,429.782,175.389,21.091,153.379
C04384=1086.412,166.970,429.760,175.391,21.093,153.379
C04385=1086.417,167.219,429.738,175.394,21.095,153.379
C04386=1086.422,167.467,429.717,175.396,21.097,153.379
C04387=1086.428,167.717,429.695,175.399,21.098,153.379
C04388=1086.433,167.965,429.674,175.401,21.100,153.379
C04389=1086.439,168.215,429.651,175.404,21.101,153.379
C04390=1086.444,168.463,429.630,175.406,21.103,153.379
C04391=1086.450,168.713,429.608,175.409,21.105,153.379
C04392=1086.455,168.961,429.587,175.411,21.107,153.379
C04393=1086.461,169.211,429.564,175.414,21.108,153.379
C04394=1086.466,169.459,429.543,175.415,21.109,153.379
C04395=1086.472,169.709,429.521,175.418,21.111,153.378
C04396=1086.478,169.958,429.499,175.420,21.113,153.379
C04397=1086.483,170.207,429.477,175.423,21.114,153.378
C04398=1086.489,170.456,429.456,175.425,21.116,153.378
C04399=1086.494,170.704,429.433,175.428,21.117,153.378
C04400=1086.500,170.953,429.412,175.430,21.119,153.378
C04401=1086.505,171.202,429.390,175.433,21.121,153.378
C04402=1086.511,171.451,429.368,175.435,21.122,153.378
C04403=1086.516,171.700,429.346,175.438,21.124,153.378
C04404=1086.522,171.949,429.325,175.440,21.125,153.378
C04405=1086.527,172.199,429.302,175.443,21.127,153.378
C04406=1086.533,172.447,429.280,175.445,21.128,153.378
C04407=1086.539,172.696,429.258,175.447,21.130,153.378
C04408=1086.544,172.945,429.236,175.450,21.132,153.378
C04409=1086.550,173.194,429.215,175.452,21.133,153.378
C04410=1086.555,173.443,429.192,175.455,21.135,153.378
C04411=1086.561,173.692,429.170,175.457,21.136,153.378
C04412=1086.566,173.941,429.148,175.460,21.138,153.378
C04413=1086.571,174.190,429.126,175.462,21.140,153.377
C04414=1086.578,174.439,429.104,175.465,21.141,153.377
C04415=1086.583,174.688,429.082,175.467,21.143,153.377
C04416=1086.589,174.937,429.060,175.470,21.144,153.377
C04417=1086.594,175.185,429.037,175.472,21.146,153.377
C04418=1086.601,175.464,429.013,175.475,21.148,153.377
C04419=1086.606,175.742,428.988,175.477,21.149,153.377
C04420=1086.613,176.020,428.963,175.481,21.151,153.377
C04421=1086.619,176.298,428.939,175.483,21.153,153.377
C04422=1086.625,176.547,428.917,175.486,21.154,153.377
C04423=1086.630,176.796,428.894,175.488,21.156,153.377
C04424=1086.636,177.045,428.873,175.491,21.158,153.377
C04425=1086.642,177.294,428.850,175.493,21.159,153.377
C04426=1086.647,177.543,428.828,175.496,21.161,153.377
C04427=1086.653,177.792,428.806,175.498,21.162,153.376
C04428=1086.659,178.041,428.783,175.501,21.164,153.376
C04429=1086.664,178.290,428.761,175.503,21.166,153.376
C04430=1086.670,178.538,428.739,175.506,21.167,153.376
C04431=1086.676,178.788,428.717,175.509,21.168,153.376
C04432=1086.681,179.036,428.694,175.511,21.170,153.376
C04433=1086.687,179.286,428.672,175.514,21.172,153.376
C04434=1086.693,179.534,428.650,175.516,21.173,153.376
C04435=1086.698,179.783,428.628,175.519,21.175,153.376
C04436=1086.704,180.032,428.605,175.521,21.176,153.376
C04437=1086.710,180.282,428.583,175.524,21.178,153.376
C04438=1086.715,180.530,428.560,175.526,21.179,153.376
C04439=1086.720,180.779,428.538,175.528,21.180,153.376
C04440=1086.727,181.028,428.516,175.531,21.182,153.375
C04441=1086.733,181.277,428.493,175.533,21.183,153.375
C04442=1086.738,181.526,428.471,175.536,21.185,153.375
C04443=1086.744,181.774,428.449,175.538,21.186,153.375
C04444=1086.749,182.024,428.426,175.541,21.188,153.375
C04445=1086.755,182.273,428.403,175.543,21.190,153.375
C04446=1086.761,182.521,428.381,175.546,21.191,153.375
C04447=1086.767,182.771,428.359,175.549,21.192,153.375
C04448=1086.773,183.020,428.336,175.551,21.194,153.375
C04449=1086.778,183.268,428.313,175.554,21.195,153.375
C04450=1086.783,183.517,428.291,175.556,21.197,153.374
C04451=1086.790,183.766,428.269,175.559,21.199,153.375
C04452=1086.795,184.015,428.246,175.561,21.200,153.374
C04453=1086.801,184.264,428.224,175.564,21.201,153.374
C04454=1086.807,184.513,428.201,175.567,21.203,153.374
C04455=1086.813,184.762,428.178,175.569,21.204,153.374
C04456=1086.819,185.011,428.156,175.572,21.206,153.374
C04457=1086.824,185.259,428.134,175.575,21.208,153.374
C04458=1086.829,185.508,428.111,175.578,21.209,153.374
C04459=1086.835,185.757,428.088,175.580,21.211,153.374
C04460=1086.841,186.006,428.065,175.583,21.213,153.374
C04461=1086.845,186.255,428.042,175.585,21.214,153.374
C04462=1086.851,186.504,428.019,175.588,21.216,153.374
C04463=1086.856,186.753,427.996,175.590,21.217,153.373
C04464=1086.862,187.002,427.973,175.593,21.219,153.373
C04465=1086.868,187.251,427.950,175.595,21.221,153.373
C04466=1086.873,187.500,427.929,175.598,21.222,153.373
C04467=1086.878,187.749,427.906,175.600,21.224,153.373
C04468=1086.884,187.997,427.883,175.603,21.225,153.373
C04469=1086.889,188.247,427.859,175.606,21.227,153.373
C04470=1086.895,188.496,427.836,175.608,21.229,153.373
C04471=1086.900,188.744,427.814,175.611,21.230,153.373
C04472=1086.906,188.993,427.791,175.613,21.231,153.373
C04473=1086.911,189.242,427.768,175.616,21.233,153.373
C04474=1086.917,189.490,427.745,175.618,21.235,153.373
C04475=1086.922,189.740,427.722,175.621,21.236,153.373
C04476=1086.928,189.989,427.699,175.623,21.238,153.373
C04477=1086.933,190.237,427.676,175.626,21.239,153.373
C04478=1086.938,190.486,427.653,175.628,21.241,153.372
C04479=1086.944,190.735,427.631,175.631,21.242,153.372
C04480=1086.950,190.984,427.608,175.633,21.244,153.372
C04481=1086.955,191.233,427.584,175.637,21.246,153.372
C04482=1086.962,191.511,427.559,175.640,21.247,153.372
C04483=1086.967,191.789,427.532,175.642,21.249,153.372
C04484=1086.973,192.066,427.507,175.645,21.251,153.372
C04485=1086.980,192.344,427.482,175.648,21.253,153.372
C04486=1086.985,192.592,427.457,175.651,21.254,153.372
C04487=1086.991,192.841,427.435,175.653,21.256,153.372
C04488=1086.997,193.090,427.412,175.656,21.257,153.372
C04489=1087.002,193.339,427.389,175.659,21.259,153.371
C04490=1087.007,193.588,427.365,175.662,21.261,153.371
C04491=1087.013,193.837,427.342,175.664,21.263,153.371
C04492=1087.019,194.086,427.319,175.667,21.264,153.371
C04493=1087.025,194.335,427.296,175.669,21.265,153.371
C04494=1087.030,194.584,427.273,175.672,21.267,153.371
C04495=1087.036,194.833,427.249,175.674,21.269,153.371
C04496=1087.041,195.081,427.226,175.677,21.270,153.371
C04497=1087.047,195.330,427.203,175.680,21.271,153.371
C04498=1087.052,195.580,427.180,175.682,21.273,153.371
C04499=1087.058,195.828,427.157,175.685,21.274,153.371
C04500=1087.064,196.077,427.133,175.687,21.276,153.371
C04501=1087.070,196.326,427.110,175.691,21.278,153.370
C04502=1087.075,196.575,427.087,175.693,21.279,153.370
C04503=1087.080,196.824,427.064,175.696,21.281,153.370
C04504=1087.086,197.072,427.040,175.698,21.282,153.370
C04505=1087.091,197.321,427.016,175.701,21.284,153.370
C04506=1087.097,197.570,426.993,175.703,21.286,153.370
C04507=1087.103,197.819,426.971,175.706,21.287,153.370
C04508=1087.109,198.067,426.947,175.709,21.288,153.370
C04509=1087.114,198.316,426.923,175.711,21.290,153.370
C04510=1087.120,198.565,426.900,175.715,21.292,153.370
C04511=1087.126,198.814,426.877,175.717,21.293,153.369
C04512=1087.131,199.063,426.853,175.720,21.295,153.369
C04513=1087.137,199.311,426.829,175.722,21.296,153.369
C04514=1087.143,199.561,426.806,175.725,21.298,153.369
C04515=1087.148,199.810,426.783,175.728,21.299,153.369
C04516=1087.154,200.058,426.759,175.730,21.301,153.369
C04517=1087.160,200.307,426.736,175.733,21.302,153.369
C04518=1087.165,200.556,426.712,175.736,21.304,153.369
C04519=1087.171,200.805,426.689,175.739,21.306,153.369
C04520=1087.176,201.054,426.665,175.741,21.307,153.369
C04521=1087.182,201.302,426.642,175.744,21.309,153.369
C04522=1087.188,201.552,426.618,175.747,21.310,153.368
C04523=1087.193,201.800,426.594,175.749,21.311,153.368
C04524=1087.199,202.049,426.571,175.752,21.313,153.368
C04525=1087.205,202.297,426.547,175.755,21.315,153.368
C04526=1087.210,202.547,426.524,175.758,21.316,153.368
C04527=1087.216,202.795,426.500,175.760,21.317,153.368
C04528=1087.221,203.044,426.477,175.763,21.319,153.368
C04529=1087.228,203.293,426.453,175.765,21.321,153.368
C04530=1087.233,203.542,426.428,175.768,21.322,153.368
C04531=1087.238,203.791,426.405,175.771,21.324,153.368
C04532=1087.244,204.039,426.381,175.774,21.325,153.367
C04533=1087.249,204.288,426.358,175.777,21.327,153.367
C04534=1087.255,204.537,426.334,175.779,21.329,153.367
C04535=1087.260,204.786,426.310,175.782,21.330,153.367
C04536=1087.266,205.034,426.286,175.784,21.332,153.367
C04537=1087.272,205.283,426.262,175.787,21.333,153.367
C04538=1087.277,205.533,426.239,175.790,21.335,153.367
C04539=1087.282,205.781,426.214,175.793,21.337,153.367
C04540=1087.289,206.029,426.191,175.796,21.338,153.367
C04541=1087.294,206.279,426.167,175.798,21.339,153.367
C04542=1087.300,206.527,426.144,175.801,21.341,153.367
C04543=1087.305,206.776,426.119,175.803,21.343,153.367
C04544=1087.311,207.025,426.095,175.807,21.345,153.366
C04545=1087.316,207.274,426.072,175.809,21.346,153.366
C04546=1087.339,208.299,425.972,175.886,21.385,153.363
C04547=1087.348,208.684,425.935,175.889,21.389,153.363
C04548=1087.357,209.069,425.897,175.894,21.393,153.363
C04549=1087.365,209.454,425.859,175.898,21.397,153.363
C04550=1087.375,209.840,425.821,175.902,21.401,153.363
C04551=1087.380,210.088,425.797,175.905,21.403,153.364
C04552=1087.385,210.337,425.773,175.907,21.405,153.364
C04553=1087.391,210.586,425.748,175.909,21.408,153.364
C04554=1087.397,210.835,425.724,175.912,21.411,153.364
C04555=1087.402,211.084,425.699,175.914,21.413,153.364
C04556=1087.408,211.332,425.674,175.918,21.415,153.364
C04557=1087.413,211.581,425.650,175.920,21.418,153.364
C04558=1087.419,211.830,425.625,175.923,21.421,153.364
C04559=1087.425,212.078,425.601,175.925,21.423,153.365
C04560=1087.430,212.328,425.577,175.927,21.425,153.365
C04561=1087.436,212.576,425.552,175.931,21.428,153.365
C04562=1087.441,212.824,425.527,175.933,21.430,153.365
C04563=1087.447,213.074,425.503,175.936,21.433,153.365
C04564=1087.453,213.322,425.478,175.938,21.435,153.365
C04565=1087.459,213.571,425.453,175.941,21.438,153.365
C04566=1087.464,213.819,425.429,175.944,21.440,153.365
C04567=1087.470,214.069,425.404,175.947,21.443,153.366
C04568=1087.476,214.317,425.379,175.949,21.445,153.366
C04569=1087.481,214.566,425.354,175.952,21.448,153.366
C04570=1087.486,214.814,425.329,175.954,21.451,153.366
C04571=1087.492,215.063,425.305,175.957,21.452,153.366
C04572=1087.498,215.312,425.280,175.960,21.455,153.366
C04573=1087.503,215.560,425.255,175.962,21.458,153.366
C04574=1087.509,215.809,425.231,175.965,21.461,153.366
C04575=1087.514,216.058,425.206,175.967,21.463,153.367
C04576=1087.520,216.307,425.180,175.970,21.465,153.367
C04577=1087.525,216.555,425.156,175.973,21.468,153.367
C04578=1087.531,216.804,425.131,175.976,21.471,153.367
C04579=1087.537,217.053,425.107,175.978,21.473,153.367
C04580=1087.543,217.301,425.081,175.981,21.476,153.367
C04581=1087.547,217.550,425.056,175.983,21.478,153.367
C04582=1087.554,217.799,425.031,175.986,21.481,153.367
C04583=1087.559,218.048,425.007,175.989,21.483,153.368
C04584=1087.565,218.296,424.981,175.992,21.486,153.368
C04585=1087.571,218.546,424.957,175.994,21.488,153.368
C04586=1087.576,218.794,424.931,175.997,21.491,153.368
C04587=1087.582,219.043,424.907,175.999,21.493,153.368
C04588=1087.587,219.291,424.882,176.002,21.496,153.368
C04589=1087.594,219.540,424.856,176.005,21.498,153.368
C04590=1087.599,219.788,424.832,176.007,21.500,153.368
C04591=1087.604,220.037,424.806,176.010,21.503,153.369
C04592=1087.611,220.286,424.781,176.012,21.505,153.369
C04593=1087.616,220.535,424.757,176.015,21.508,153.369
C04594=1087.622,220.783,424.731,176.018,21.510,153.369
C04595=1087.627,221.032,424.706,176.021,21.513,153.369
C04596=1087.633,221.281,424.681,176.023,21.515,153.369
C04597=1087.639,221.529,424.656,176.026,21.518,153.369
C04598=1087.644,221.778,424.630,176.029,21.520,153.369
C04599=1087.653,222.167,424.592,176.033,21.524,153.370
C04600=1087.662,222.557,424.552,176.037,21.528,153.370
C04601=1087.670,222.945,424.512,176.042,21.532,153.370
C04602=1087.679,223.334,424.472,176.045,21.536,153.370
C04603=1087.684,223.583,424.447,176.048,21.539,153.370
C04604=1087.690,223.831,424.422,176.051,21.541,153.371
C04605=1087.696,224.081,424.397,176.054,21.544,153.371
C04606=1087.701,224.329,424.371,176.056,21.546,153.371
C04607=1087.707,224.578,424.346,176.059,21.549,153.371
C04608=1087.713,224.826,424.320,176.061,21.551,153.371
C04609=1087.719,225.074,424.295,176.064,21.554,153.371
C04610=1087.724,225.323,424.269,176.067,21.557,153.371
C04611=1087.730,225.572,424.244,176.070,21.559,153.371
C04612=1087.735,225.821,424.219,176.073,21.562,153.371
C04613=1087.741,226.070,424.194,176.075,21.564,153.372
C04614=1087.746,226.319,424.168,176.078,21.567,153.372
C04615=1087.752,226.567,424.143,176.080,21.569,153.372
C04616=1087.758,226.816,424.117,176.084,21.572,153.372
C04617=1087.764,227.064,424.092,176.086,21.574,153.372
C04618=1087.769,227.313,424.066,176.089,21.577,153.372
C04619=1087.775,227.561,424.041,176.091,21.579,153.372
C04620=1087.780,227.810,424.015,176.094,21.582,153.373
C04621=1087.786,228.059,423.989,176.097,21.584,153.373
C04622=1087.791,228.307,423.964,176.100,21.587,153.373
C04623=1087.797,228.556,423.938,176.102,21.589,153.373
C04624=1087.803,228.805,423.912,176.105,21.592,153.373
C04625=1087.808,229.054,423.887,176.108,21.595,153.373
C04626=1087.815,229.302,423.861,176.111,21.597,153.373
C04627=1087.820,229.550,423.835,176.114,21.600,153.373
C04628=1087.826,229.799,423.810,176.116,21.602,153.374
C04629=1087.832,230.048,423.784,176.119,21.605,153.374
C04630=1087.837,230.297,423.758,176.121,21.607,153.374
C04631=1087.843,230.545,423.733,176.124,21.610,153.374
C04632=1087.848,230.794,423.707,176.127,21.612,153.374
C04633=1087.854,231.043,423.681,176.130,21.615,153.374
C04634=1087.860,231.291,423.655,176.133,21.618,153.374
C04635=1087.866,231.540,423.629,176.135,21.620,153.374
C04636=1087.870,231.788,423.603,176.138,21.623,153.375
C04637=1087.876,232.037,423.577,176.141,21.625,153.375
C04638=1087.882,232.285,423.551,176.144,21.628,153.375
C04639=1087.888,232.534,423.525,176.146,21.630,153.375
C04640=1087.893,232.783,423.499,176.149,21.633,153.375
C04641=1087.898,233.031,423.474,176.152,21.636,153.375
C04642=1087.905,233.279,423.448,176.154,21.638,153.375
C04643=1087.910,233.528,423.422,176.157,21.641,153.376
C04644=1087.916,233.777,423.396,176.160,21.643,153.376
C04645=1087.921,234.026,423.369,176.163,21.646,153.376
C04646=1087.927,234.275,423.343,176.165,21.648,153.376
C04647=1087.932,234.523,423.318,176.168,21.651,153.376
C04648=1087.938,234.771,423.292,176.171,21.654,153.376
C04649=1087.944,235.020,423.266,176.173,21.656,153.376
C04650=1087.949,235.269,423.240,176.176,21.659,153.376
C04651=1087.958,235.649,423.199,176.180,21.663,153.377
C04652=1087.966,236.030,423.160,176.185,21.667,153.377
C04653=1087.975,236.410,423.119,176.189,21.670,153.377
C04654=1087.984,236.790,423.080,176.193,21.675,153.377
C04655=1087.989,237.039,423.054,176.196,21.677,153.377
C04656=1087.995,237.287,423.027,176.199,21.680,153.378
C04657=1088.000,237.536,423.001,176.202,21.683,153.378
C04658=1088.006,237.784,422.974,176.204,21.685,153.378
C04659=1088.012,238.033,422.949,176.207,21.688,153.378
C04660=1088.017,238.282,422.922,176.210,21.690,153.378
C04661=1088.023,238.531,422.896,176.213,21.693,153.378
C04662=1088.029,238.779,422.869,176.216,21.695,153.378
C04663=1088.034,239.028,422.843,176.218,21.698,153.379
C04664=1088.040,239.276,422.817,176.221,21.701,153.379
C04665=1088.046,239.525,422.790,176.223,21.703,153.379
C04666=1088.051,239.774,422.764,176.226,21.706,153.379
C04667=1088.057,240.022,422.737,176.230,21.708,153.379
C04668=1088.063,240.271,422.711,176.232,21.711,153.379
C04669=1088.068,240.520,422.685,176.235,21.713,153.379
C04670=1088.074,240.768,422.658,176.238,21.716,153.379
C04671=1088.080,241.016,422.632,176.240,21.719,153.380
C04672=1088.085,241.265,422.606,176.243,21.721,153.380
C04673=1088.091,241.514,422.579,176.246,21.724,153.380
C04674=1088.097,241.762,422.552,176.249,21.727,153.380
C04675=1088.102,242.011,422.526,176.252,21.729,153.380
C04676=1088.108,242.259,422.500,176.254,21.731,153.380
C04677=1088.114,242.508,422.473,176.257,21.734,153.380
C04678=1088.120,242.756,422.447,176.260,21.737,153.381
C04679=1088.125,243.004,422.420,176.263,21.739,153.381
C04680=1088.131,243.253,422.394,176.266,21.742,153.381
C04681=1088.137,243.502,422.367,176.269,21.745,153.381
C04682=1088.142,243.750,422.340,176.271,21.747,153.381
C04683=1088.147,243.999,422.313,176.274,21.750,153.381
C04684=1088.153,244.247,422.287,176.276,21.753,153.382
C04685=1088.159,244.495,422.260,176.279,21.755,153.382
C04686=1088.164,244.744,422.233,176.282,21.758,153.382
C04687=1088.169,244.993,422.207,176.285,21.761,153.382
C04688=1088.175,245.241,422.180,176.288,21.763,153.382
C04689=1088.181,245.490,422.154,176.291,21.766,153.382
C04690=1088.187,245.738,422.127,176.293,21.768,153.382
C04691=1088.192,245.987,422.100,176.296,21.771,153.382
C04692=1088.198,246.235,422.073,176.299,21.774,153.383
C04693=1088.203,246.484,422.046,176.302,21.776,153.383
C04694=1088.209,246.732,422.020,176.305,21.779,153.383
C04695=1088.215,246.981,421.992,176.308,21.782,153.383
C04696=1088.221,247.230,421.966,176.310,21.784,153.383
C04697=1088.226,247.478,421.939,176.313,21.787,153.383
C04698=1088.231,247.727,421.912,176.316,21.790,153.384
C04699=1088.237,247.975,421.885,176.318,21.792,153.384
C04700=1088.242,248.224,421.858,176.322,21.795,153.384
C04701=1088.248,248.472,421.831,176.325,21.798,153.384
C04702=1088.253,248.720,421.803,176.327,21.800,153.384
C04703=1088.262,249.094,421.763,176.332,21.805,153.384
C04704=1088.270,249.468,421.722,176.335,21.808,153.385
C04705=1088.278,249.841,421.682,176.340,21.813,153.385
C04706=1088.286,250.214,421.640,176.344,21.817,153.385
C04707=1088.292,250.463,421.614,176.347,21.820,153.385
C04708=1088.298,250.712,421.586,176.350,21.823,153.386
C04709=1088.304,250.960,421.560,176.353,21.825,153.386
C04710=1088.309,251.209,421.533,176.355,21.828,153.386
C04711=1088.315,251.457,421.505,176.358,21.831,153.386
C04712=1088.320,251.705,421.478,176.361,21.833,153.386
C04713=1088.326,251.954,421.451,176.363,21.836,153.386
C04714=1088.331,252.202,421.423,176.367,21.839,153.387
C04715=1088.337,252.451,421.396,176.370,21.841,153.387
C04716=1088.342,252.700,421.369,176.373,21.844,153.387
C04717=1088.348,252.947,421.342,176.375,21.847,153.387
C04718=1088.353,253.196,421.314,176.378,21.849,153.387
C04719=1088.359,253.444,421.288,176.381,21.852,153.387
C04720=1088.365,253.693,421.259,176.383,21.855,153.387
C04721=1088.371,253.942,421.233,176.386,21.857,153.388
C04722=1088.376,254.190,421.205,176.390,21.860,153.388
C04723=1088.382,254.438,421.178,176.393,21.863,153.388
C04724=1088.388,254.687,421.150,176.395,21.865,153.388
C04725=1088.393,254.935,421.122,176.398,21.868,153.388
C04726=1088.399,255.184,421.096,176.401,21.871,153.388
C04727=1088.404,255.432,421.068,176.403,21.873,153.389
C04728=1088.411,255.681,421.041,176.406,21.876,153.389
C04729=1088.416,255.929,421.013,176.410,21.879,153.389
C04730=1088.422,256.177,420.986,176.413,21.882,153.389
C04731=1088.428,256.426,420.958,176.415,21.884,153.389
C04732=1088.433,256.675,420.931,176.418,21.887,153.389
C04733=1088.439,256.922,420.903,176.421,21.890,153.390
C04734=1088.444,257.172,420.876,176.423,21.892,153.390
C04735=1088.450,257.419,420.848,176.426,21.895,153.390
C04736=1088.455,257.668,420.821,176.429,21.898,153.390
C04737=1088.461,257.917,420.793,176.433,21.901,153.390
C04738=1088.467,258.165,420.765,176.435,21.903,153.390
C04739=1088.473,258.413,420.738,176.438,21.906,153.390
C04740=1088.478,258.662,420.710,176.441,21.909,153.391
C04741=1088.485,258.910,420.682,176.444,21.912,153.391
C04742=1088.490,259.158,420.655,176.446,21.914,153.391
C04743=1088.496,259.407,420.627,176.449,21.917,153.391
C04744=1088.502,259.655,420.600,176.453,21.920,153.391
C04745=1088.507,259.904,420.572,176.456,21.922,153.391
C04746=1088.513,260.152,420.544,176.458,21.925,153.392
C04747=1088.519,260.400,420.517,176.461,21.927,153.392
C04748=1088.525,260.649,420.488,176.464,21.930,153.392
C04749=1088.530,260.898,420.461,176.467,21.933,153.392
C04750=1088.536,261.146,420.433,176.469,21.935,153.392
C04751=1088.542,261.394,420.405,176.473,21.938,153.392
C04752=1088.547,261.642,420.377,176.476,21.941,153.393
C04753=1088.553,261.891,420.350,176.479,21.944,153.393
C04754=1088.559,262.139,420.322,176.481,21.946,153.393
C04755=1088.567,262.510,420.280,176.486,21.951,153.393
C04756=1088.576,262.881,420.239,176.490,21.955,153.393
C04757=1088.585,263.251,420.197,176.494,21.959,153.394
C04758=1088.593,263.622,420.155,176.499,21.963,153.394
C04759=1088.599,263.870,420.127,176.502,21.966,153.394
C04760=1088.605,264.118,420.100,176.504,21.968,153.394
C04761=1088.611,264.367,420.071,176.507,21.971,153.394
C04762=1088.616,264.615,420.043,176.510,21.974,153.395
C04763=1088.622,264.864,420.016,176.513,21.977,153.395
C04764=1088.627,265.112,419.988,176.516,21.980,153.395
C04765=1088.634,265.360,419.959,176.519,21.982,153.395
C04766=1088.639,265.608,419.931,176.522,21.985,153.395
C04767=1088.645,265.857,419.902,176.525,21.988,153.395
C04768=1088.650,266.105,419.874,176.528,21.991,153.396
C04769=1088.656,266.354,419.846,176.530,21.993,153.396
C04770=1088.662,266.602,419.818,176.533,21.996,153.396
C04771=1088.668,266.851,419.790,176.536,21.999,153.396
C04772=1088.673,267.099,419.762,176.539,22.002,153.396
C04773=1088.679,267.348,419.734,176.542,22.005,153.396
C04774=1088.684,267.596,419.706,176.544,22.007,153.397
C04775=1088.690,267.844,419.677,176.547,22.010,153.397
C04776=1088.696,268.092,419.649,176.551,22.013,153.397
C04777=1088.702,268.341,419.620,176.554,22.016,153.397
C04778=1088.707,268.589,419.592,176.557,22.019,153.397
C04779=1088.713,268.837,419.564,176.560,22.021,153.398
C04780=1088.718,269.085,419.536,176.562,22.024,153.398
C04781=1088.724,269.334,419.506,176.565,22.027,153.398
C04782=1088.729,269.582,419.478,176.568,22.030,153.398
C04783=1088.735,269.831,419.450,176.571,22.033,153.398
C04784=1088.741,270.079,419.422,176.574,22.035,153.398
C04785=1088.747,270.327,419.393,176.576,22.038,153.399
C04786=1088.753,270.576,419.365,176.580,22.041,153.399
C04787=1088.758,270.824,419.337,176.583,22.044,153.399
C04788=1088.764,271.072,419.307,176.586,22.047,153.399
C04789=1088.769,271.320,419.279,176.589,22.050,153.400
C04790=1088.775,271.569,419.251,176.592,22.053,153.400
C04791=1088.781,271.817,419.222,176.594,22.055,153.400
C04792=1088.786,272.065,419.194,176.597,22.058,153.400
C04793=1088.793,272.313,419.165,176.600,22.061,153.400
C04794=1088.797,272.562,419.136,176.603,22.064,153.400
C04795=1088.803,272.810,419.108,176.606,22.067,153.401
C04796=1088.809,273.059,419.079,176.609,22.069,153.401
C04797=1088.815,273.307,419.051,176.611,22.073,153.401
C04798=1088.820,273.555,419.021,176.615,22.075,153.401
C04799=1088.826,273.804,418.993,176.618,22.078,153.401
C04800=1088.832,274.051,418.964,176.621,22.081,153.402
C04801=1088.838,274.300,418.936,176.624,22.084,153.402
C04802=1088.843,274.548,418.906,176.627,22.087,153.402
C04803=1088.849,274.796,418.878,176.629,22.089,153.402
C04804=1088.855,275.045,418.849,176.632,22.093,153.402
C04805=1088.860,275.293,418.821,176.635,22.095,153.403
C04806=1088.866,275.541,418.792,176.638,22.098,153.403
C04807=1088.874,275.915,418.748,176.643,22.103,153.403
C04808=1088.883,276.288,418.705,176.647,22.107,153.403
C04809=1088.891,276.662,418.661,176.651,22.111,153.404
C04810=1088.900,277.035,418.617,176.656,22.116,153.404
C04811=1088.906,277.283,418.589,176.659,22.119,153.404
C04812=1088.911,277.532,418.560,176.662,22.122,153.404
C04813=1088.917,277.780,418.531,176.665,22.125,153.405
C04814=1088.923,278.029,418.502,176.668,22.128,153.405
C04815=1088.928,278.276,418.473,176.671,22.131,153.405
C04816=1088.934,278.525,418.443,176.673,22.133,153.405
C04817=1088.940,278.773,418.414,176.676,22.136,153.406
C04818=1088.945,279.021,418.386,176.679,22.139,153.406
C04819=1088.951,279.269,418.357,176.682,22.142,153.406
C04820=1088.956,279.518,418.327,176.685,22.145,153.406
C04821=1088.963,279.766,418.298,176.688,22.148,153.406
C04822=1088.968,280.014,418.269,176.691,22.151,153.407
C04823=1088.974,280.262,418.240,176.694,22.154,153.407
C04824=1088.980,280.510,418.212,176.696,22.157,153.407
C04825=1088.985,280.759,418.182,176.700,22.160,153.407
C04826=1088.991,281.007,418.152,176.703,22.162,153.407
C04827=1088.996,281.255,418.124,176.706,22.166,153.408
C04828=1089.002,281.503,418.094,176.709,22.168,153.408
C04829=1089.008,281.751,418.065,176.712,22.172,153.408
C04830=1089.014,282.000,418.035,176.715,22.175,153.408
C04831=1089.019,282.247,418.006,176.718,22.178,153.409
C04832=1089.025,282.496,417.977,176.721,22.181,153.409
C04833=1089.030,282.744,417.947,176.724,22.184,153.409
C04834=1089.036,282.993,417.918,176.726,22.186,153.409
C04835=1089.042,283.241,417.889,176.729,22.190,153.410
C04836=1089.047,283.488,417.859,176.732,22.192,153.410
C04837=1089.053,283.737,417.830,176.735,22.196,153.410
C04838=1089.059,283.985,417.801,176.738,22.198,153.410
C04839=1089.064,284.233,417.771,176.741,22.202,153.410
C04840=1089.070,284.482,417.741,176.744,22.204,153.411
C04841=1089.076,284.730,417.712,176.747,22.208,153.411
C04842=1089.081,284.977,417.682,176.750,22.211,153.411
C04843=1089.087,285.226,417.653,176.753,22.214,153.411
C04844=1089.092,285.474,417.623,176.756,22.217,153.412
C04845=1089.099,285.722,417.594,176.759,22.220,153.412
C04846=1089.104,285.971,417.564,176.761,22.223,153.412
C04847=1089.110,286.219,417.535,176.764,22.226,153.412
C04848=1089.115,286.467,417.504,176.767,22.229,153.413
C04849=1089.122,286.715,417.475,176.770,22.232,153.413
C04850=1089.127,286.963,417.446,176.773,22.235,153.413
C04851=1089.132,287.211,417.417,176.777,22.238,153.413
C04852=1089.138,287.459,417.386,176.779,22.241,153.414
C04853=1089.144,287.707,417.357,176.783,22.244,153.414
C04854=1089.150,287.956,417.328,176.785,22.247,153.414
C04855=1089.155,288.203,417.297,176.789,22.250,153.414
C04856=1089.161,288.452,417.268,176.792,22.253,153.414
C04857=1089.167,288.700,417.238,176.795,22.256,153.415
C04858=1089.173,288.948,417.208,176.798,22.259,153.415
C04859=1089.182,289.331,417.162,176.802,22.264,153.415
C04860=1089.190,289.715,417.116,176.807,22.268,153.416
C04861=1089.199,290.097,417.070,176.811,22.273,153.416
C04862=1089.208,290.480,417.024,176.816,22.278,153.416
C04863=1089.214,290.728,416.994,176.819,22.281,153.417
C04864=1089.220,290.976,416.964,176.822,22.284,153.417
C04865=1089.225,291.224,416.934,176.825,22.287,153.417
C04866=1089.231,291.472,416.904,176.828,22.290,153.417
C04867=1089.237,291.720,416.874,176.831,22.293,153.418
C04868=1089.242,291.969,416.844,176.834,22.296,153.418
C04869=1089.248,292.216,416.814,176.837,22.300,153.418
C04870=1089.254,292.465,416.784,176.840,22.303,153.419
C04871=1089.259,292.713,416.754,176.843,22.306,153.419
C04872=1089.265,292.961,416.724,176.846,22.309,153.419
C04873=1089.271,293.209,416.694,176.849,22.312,153.419
C04874=1089.277,293.457,416.664,176.852,22.315,153.419
C04875=1089.282,293.705,416.634,176.855,22.318,153.420
C04876=1089.288,293.953,416.604,176.858,22.322,153.420
C04877=1089.294,294.201,416.573,176.860,22.325,153.420
C04878=1089.298,294.450,416.543,176.864,22.328,153.421
C04879=1089.304,294.697,416.513,176.867,22.331,153.421
C04880=1089.310,294.945,416.482,176.870,22.334,153.421
C04881=1089.316,295.193,416.452,176.872,22.337,153.421
C04882=1089.322,295.442,416.422,176.876,22.340,153.422
C04883=1089.328,295.690,416.392,176.879,22.343,153.422
C04884=1089.334,295.938,416.361,176.881,22.347,153.422
C04885=1089.340,296.186,416.331,176.884,22.350,153.422
C04886=1089.345,296.434,416.301,176.887,22.353,153.423
C04887=1089.351,296.682,416.271,176.890,22.356,153.423
C04888=1089.356,296.930,416.240,176.893,22.359,153.423
C04889=1089.362,297.178,416.210,176.896,22.363,153.424
C04890=1089.368,297.426,416.179,176.899,22.366,153.424
C04891=1089.373,297.674,416.149,176.902,22.369,153.424
C04892=1089.380,297.922,416.118,176.905,22.372,153.424
C04893=1089.385,298.171,416.088,176.908,22.375,153.425
C04894=1089.390,298.419,416.058,176.911,22.378,153.425
C04895=1089.396,298.666,416.027,176.914,22.382,153.425
C04896=1089.401,298.915,415.996,176.917,22.385,153.426
C04897=1089.407,299.162,415.966,176.920,22.388,153.426
C04898=1089.412,299.411,415.935,176.923,22.391,153.426
C04899=1089.418,299.658,415.905,176.926,22.395,153.427
C04900=1089.424,299.906,415.874,176.929,22.398,153.427
C04901=1089.429,300.154,415.844,176.932,22.402,153.427
C04902=1089.435,300.403,415.813,176.935,22.405,153.427
C04903=1089.440,300.651,415.782,176.938,22.408,153.428
C04904=1089.447,300.898,415.751,176.941,22.412,153.428
C04905=1089.452,301.146,415.720,176.944,22.415,153.428
C04906=1089.457,301.394,415.689,176.947,22.418,153.429
C04907=1089.463,301.642,415.659,176.950,22.422,153.429
C04908=1089.468,301.890,415.628,176.953,22.425,153.429
C04909=1089.475,302.139,415.597,176.956,22.428,153.430
C04910=1089.480,302.387,415.567,176.959,22.431,153.430
C04911=1089.489,302.784,415.517,176.964,22.437,153.430
C04912=1089.498,303.181,415.468,176.969,22.442,153.431
C04913=1089.507,303.577,415.419,176.973,22.447,153.431
C04914=1089.516,303.974,415.369,176.978,22.453,153.432
C04915=1089.522,304.222,415.338,176.981,22.456,153.432
C04916=1089.528,304.470,415.307,176.984,22.459,153.432
C04917=1089.533,304.719,415.276,176.987,22.463,153.433
C04918=1089.539,304.966,415.245,176.990,22.466,153.433
C04919=1089.544,305.214,415.214,176.993,22.469,153.433
C04920=1089.550,305.462,415.183,176.997,22.473,153.434
C04921=1089.556,305.710,415.152,177.000,22.476,153.434
C04922=1089.562,305.958,415.121,177.003,22.480,153.434
C04923=1089.567,306.207,415.090,177.006,22.483,153.435
C04924=1089.573,306.454,415.059,177.009,22.486,153.435
C04925=1089.578,306.702,415.028,177.011,22.489,153.435
C04926=1089.585,306.950,414.996,177.014,22.493,153.436
C04927=1089.590,307.198,414.965,177.017,22.496,153.436
C04928=1089.596,307.445,414.934,177.020,22.500,153.436
C04929=1089.601,307.693,414.903,177.023,22.503,153.437
C04930=1089.607,307.942,414.871,177.027,22.507,153.437
C04931=1089.613,308.189,414.841,177.030,22.510,153.437
C04932=1089.619,308.438,414.809,177.033,22.513,153.438
C04933=1089.625,308.685,414.779,177.036,22.516,153.438
C04934=1089.630,308.933,414.747,177.039,22.520,153.438
C04935=1089.636,309.182,414.716,177.042,22.523,153.439
C04936=1089.642,309.429,414.685,177.045,22.527,153.439
C04937=1089.648,309.678,414.653,177.047,22.530,153.439
C04938=1089.653,309.925,414.622,177.051,22.534,153.439
C04939=1089.659,310.172,414.591,177.054,22.537,153.440
C04940=1089.665,310.421,414.559,177.057,22.540,153.440
C04941=1089.671,310.669,414.528,177.060,22.544,153.441
C04942=1089.677,310.917,414.496,177.063,22.547,153.441
C04943=1089.682,311.165,414.465,177.066,22.551,153.441
C04944=1089.688,311.413,414.433,177.069,22.554,153.442
C04945=1089.694,311.660,414.402,177.072,22.557,153.442
C04946=1089.700,311.908,414.370,177.076,22.561,153.442
C04947=1089.706,312.157,414.339,177.079,22.564,153.442
C04948=1089.712,312.405,414.308,177.081,22.568,153.443
C04949=1089.718,312.652,414.276,177.084,22.571,153.443
C04950=1089.724,312.900,414.244,177.087,22.574,153.444
C04951=1089.729,313.148,414.214,177.090,22.578,153.444
C04952=1089.735,313.396,414.182,177.093,22.581,153.444
C04953=1089.741,313.644,414.150,177.097,22.585,153.445
C04954=1089.747,313.892,414.118,177.100,22.588,153.445
C04955=1089.753,314.139,414.087,177.103,22.592,153.445
C04956=1089.759,314.387,414.055,177.106,22.595,153.446
C04957=1089.765,314.636,414.023,177.108,22.598,153.446
C04958=1089.770,314.883,413.991,177.111,22.602,153.446
C04959=1089.777,315.132,413.961,177.114,22.605,153.447
C04960=1089.781,315.379,413.928,177.118,22.609,153.447
C04961=1089.787,315.628,413.896,177.121,22.613,153.447
C04962=1089.793,315.875,413.865,177.124,22.616,153.448
C04963=1089.802,316.275,413.813,177.129,22.622,153.448
C04964=1089.811,316.675,413.761,177.133,22.628,153.449
C04965=1089.821,317.074,413.710,177.138,22.634,153.450
C04966=1089.829,317.474,413.659,177.143,22.640,153.450
C04967=1089.835,317.722,413.627,177.146,22.643,153.451
C04968=1089.841,317.970,413.594,177.149,22.647,153.451
C04969=1089.846,318.218,413.562,177.152,22.651,153.452
C04970=1089.852,318.466,413.530,177.155,22.654,153.452
C04971=1089.857,318.713,413.498,177.158,22.658,153.452
C04972=1089.863,318.961,413.466,177.161,22.662,153.453
C04973=1089.869,319.209,413.435,177.164,22.665,153.453
C04974=1089.874,319.458,413.402,177.167,22.669,153.454
C04975=1089.880,319.705,413.369,177.170,22.673,153.454
C04976=1089.886,319.953,413.338,177.173,22.677,153.454
C04977=1089.892,320.201,413.306,177.176,22.680,153.455
C04978=1089.897,320.448,413.274,177.179,22.683,153.455
C04979=1089.903,320.696,413.241,177.182,22.687,153.456
C04980=1089.909,320.944,413.209,177.185,22.691,153.456
C04981=1089.914,321.192,413.177,177.188,22.695,153.456
C04982=1089.920,321.440,413.145,177.191,22.699,153.457
C04983=1089.926,321.688,413.112,177.194,22.702,153.457
C04984=1089.931,321.936,413.080,177.198,22.706,153.458
C04985=1089.937,322.184,413.048,177.200,22.710,153.458
C04986=1089.943,322.431,413.015,177.203,22.714,153.459
C04987=1089.949,322.679,412.984,177.206,22.717,153.459
C04988=1089.954,322.927,412.950,177.210,22.721,153.459
C04989=1089.960,323.175,412.918,177.213,22.725,153.460
C04990=1089.966,323.423,412.886,177.215,22.728,153.460
C04991=1089.972,323.670,412.854,177.218,22.732,153.461
C04992=1089.977,323.919,412.821,177.221,22.736,153.461
C04993=1089.983,324.166,412.788,177.225,22.740,153.461
C04994=1089.989,324.414,412.756,177.228,22.744,153.462
C04995=1089.994,324.662,412.723,177.230,22.747,153.462
C04996=1090.000,324.910,412.691,177.233,22.750,153.463
C04997=1090.007,325.157,412.659,177.237,22.755,153.463
C04998=1090.012,325.406,412.626,177.240,22.758,153.463
C04999=1090.018,325.654,412.593,177.243,22.762,153.464
C05000=1090.024,325.900,412.561,177.245,22.766,153.464
C05001=1090.030,326.149,412.529,177.249,22.770,153.465
C05002=1090.035,326.397,412.496,177.252,22.773,153.465
C05003=1090.041,326.645,412.464,177.255,22.777,153.466
C05004=1090.047,326.893,412.430,177.258,22.781,153.466
C05005=1090.053,327.140,412.398,177.261,22.785,153.467
C05006=1090.059,327.388,412.366,177.264,22.789,153.467
C05007=1090.064,327.636,412.332,177.267,22.792,153.467
C05008=1090.070,327.883,412.300,177.270,22.797,153.468
C05009=1090.077,328.131,412.267,177.273,22.800,153.468
C05010=1090.082,328.379,412.234,177.276,22.804,153.469
C05011=1090.088,328.627,412.202,177.280,22.808,153.469
C05012=1090.094,328.875,412.168,177.283,22.812,153.470
C05013=1090.100,329.123,412.136,177.285,22.815,153.470
C05014=1090.106,329.370,412.104,177.288,22.819,153.471
C05015=1090.115,329.763,412.051,177.293,22.826,153.471
C05016=1090.124,330.156,411.999,177.298,22.832,153.472
C05017=1090.134,330.550,411.947,177.303,22.837,153.473
C05018=1090.143,330.942,411.895,177.308,22.844,153.473
C05019=1090.149,331.189,411.862,177.311,22.848,153.474
C05020=1090.155,331.437,411.829,177.314,22.851,153.474
C05021=1090.161,331.685,411.796,177.317,22.855,153.475
C05022=1090.167,331.933,411.762,177.320,22.859,153.475
C05023=1090.173,332.180,411.730,177.323,22.863,153.476
C05024=1090.179,332.428,411.696,177.327,22.867,153.476
C05025=1090.184,332.676,411.663,177.329,22.872,153.477
C05026=1090.190,332.924,411.630,177.332,22.875,153.477
C05027=1090.196,333.172,411.597,177.336,22.879,153.478
C05028=1090.201,333.419,411.564,177.338,22.883,153.478
C05029=1090.207,333.667,411.531,177.342,22.888,153.479
C05030=1090.213,333.914,411.498,177.345,22.892,153.479
C05031=1090.218,334.162,411.465,177.348,22.895,153.480
C05032=1090.224,334.410,411.431,177.351,22.900,153.480
C05033=1090.230,334.658,411.397,177.354,22.904,153.481
C05034=1090.236,334.905,411.364,177.357,22.908,153.481
C05035=1090.242,335.153,411.331,177.360,22.912,153.482
C05036=1090.247,335.401,411.298,177.363,22.916,153.482
C05037=1090.253,335.649,411.264,177.366,22.920,153.483
C05038=1090.258,335.897,411.231,177.369,22.924,153.483
C05039=1090.265,336.144,411.198,177.372,22.928,153.484
C05040=1090.270,336.392,411.164,177.376,22.933,153.484
C05041=1090.277,336.640,411.131,177.378,22.936,153.485
C05042=1090.282,336.888,411.097,177.381,22.940,153.485
C05043=1090.288,337.135,411.063,177.385,22.945,153.486
C05044=1090.294,337.383,411.030,177.387,22.949,153.486
C05045=1090.300,337.630,410.996,177.391,22.953,153.487
C05046=1090.306,337.878,410.963,177.394,22.957,153.487
C05047=1090.311,338.126,410.930,177.396,22.961,153.488
C05048=1090.317,338.373,410.896,177.400,22.965,153.488
C05049=1090.323,338.621,410.862,177.403,22.969,153.489
C05050=1090.328,338.869,410.829,177.406,22.974,153.489
C05051=1090.334,339.116,410.795,177.409,22.978,153.490
C05052=1090.340,339.364,410.762,177.412,22.982,153.491
C05053=1090.346,339.612,410.727,177.415,22.986,153.491
C05054=1090.352,339.860,410.694,177.418,22.990,153.492
C05055=1090.358,340.108,410.660,177.421,22.995,153.492
C05056=1090.363,340.355,410.626,177.424,22.999,153.493
C05057=1090.369,340.603,410.592,177.428,23.004,153.493
C05058=1090.375,340.851,410.559,177.430,23.007,153.494
C05059=1090.380,341.098,410.525,177.433,23.012,153.494
C05060=1090.386,341.345,410.491,177.437,23.016,153.495
C05061=1090.392,341.594,410.457,177.439,23.020,153.496
C05062=1090.398,341.841,410.423,177.443,23.025,153.496
C05063=1090.404,342.089,410.390,177.445,23.029,153.497
C05064=1090.410,342.336,410.356,177.449,23.034,153.497
C05065=1090.416,342.584,410.322,177.452,23.038,153.498
C05066=1090.421,342.831,410.288,177.455,23.042,153.498
C05067=1090.431,343.219,410.235,177.460,23.049,153.499
C05068=1090.440,343.606,410.182,177.465,23.056,153.500
C05069=1090.449,343.993,410.129,177.470,23.062,153.501
C05070=1090.458,344.380,410.076,177.474,23.069,153.502
C05071=1090.464,344.627,410.042,177.477,23.073,153.503
C05072=1090.470,344.875,410.007,177.480,23.078,153.503
C05073=1090.475,345.123,409.973,177.483,23.082,153.504
C05074=1090.481,345.370,409.939,177.486,23.087,153.504
C05075=1090.487,345.617,409.905,177.489,23.091,153.505
C05076=1090.493,345.866,409.871,177.492,23.095,153.506
C05077=1090.498,346.113,409.836,177.495,23.100,153.506
C05078=1090.504,346.361,409.802,177.498,23.104,153.507
C05079=1090.510,346.608,409.768,177.502,23.109,153.507
C05080=1090.517,346.856,409.734,177.504,23.113,153.508
C05081=1090.522,347.103,409.699,177.508,23.118,153.509
C05082=1090.528,347.351,409.665,177.511,23.123,153.509
C05083=1090.534,347.598,409.631,177.514,23.127,153.510
C05084=1090.539,347.846,409.596,177.517,23.132,153.510
C05085=1090.545,348.094,409.562,177.520,23.136,153.511
C05086=1090.551,348.341,409.528,177.523,23.141,153.512
C05087=1090.557,348.589,409.493,177.526,23.145,153.512
C05088=1090.563,348.836,409.459,177.529,23.150,153.513
C05089=1090.569,349.083,409.424,177.532,23.154,153.514
C05090=1090.574,349.331,409.389,177.535,23.159,153.514
C05091=1090.580,349.579,409.355,177.538,23.163,153.515
C05092=1090.586,349.826,409.321,177.542,23.168,153.516
C05093=1090.592,350.074,409.286,177.544,23.172,153.516
C05094=1090.598,350.322,409.252,177.548,23.177,153.517
C05095=1090.603,350.569,409.216,177.550,23.181,153.517
C05096=1090.610,350.817,409.182,177.554,23.186,153.518
C05097=1090.615,351.064,409.147,177.557,23.191,153.519
C05098=1090.621,351.311,409.113,177.560,23.195,153.519
C05099=1090.627,351.559,409.078,177.563,23.200,153.520
C05100=1090.633,351.806,409.044,177.566,23.205,153.521
C05101=1090.639,352.054,409.009,177.569,23.210,153.521
C05102=1090.644,352.301,408.974,177.572,23.214,153.522
C05103=1090.651,352.549,408.939,177.575,23.219,153.523
C05104=1090.656,352.797,408.905,177.579,23.224,153.523
C05105=1090.662,353.044,408.870,177.581,23.228,153.524
C05106=1090.668,353.292,408.835,177.585,23.233,153.525
C05107=1090.674,353.539,408.800,177.587,23.237,153.525
C05108=1090.680,353.787,408.765,177.591,23.242,153.526
C05109=1090.686,354.034,408.731,177.594,23.247,153.527
C05110=1090.692,354.282,408.695,177.596,23.252,153.528
C05111=1090.697,354.529,408.661,177.600,23.257,153.528
C05112=1090.703,354.776,408.626,177.602,23.262,153.529
C05113=1090.709,355.024,408.591,177.606,23.267,153.530
C05114=1090.714,355.271,408.556,177.609,23.271,153.530
C05115=1090.721,355.519,408.520,177.612,23.276,153.531
C05116=1090.726,355.766,408.486,177.615,23.281,153.532
C05117=1090.732,356.014,408.450,177.619,23.286,153.532
C05118=1090.738,356.261,408.416,177.621,23.290,153.533
C05119=1090.747,356.651,408.361,177.626,23.298,153.534
C05120=1090.756,357.040,408.305,177.631,23.306,153.535
C05121=1090.765,357.431,408.249,177.636,23.314,153.536
C05122=1090.775,357.820,408.194,177.640,23.321,153.538
C05123=1090.781,358.067,408.159,177.644,23.326,153.538
C05124=1090.787,358.314,408.123,177.647,23.331,153.539
C05125=1090.793,358.563,408.088,177.649,23.336,153.540
C05126=1090.798,358.810,408.053,177.653,23.341,153.541
C05127=1090.805,359.057,408.018,177.656,23.346,153.541
C05128=1090.810,359.304,407.983,177.659,23.351,153.542
C05129=1090.816,359.552,407.947,177.662,23.356,153.543
C05130=1090.822,359.799,407.911,177.665,23.361,153.544
C05131=1090.828,360.047,407.877,177.668,23.366,153.544
C05132=1090.834,360.294,407.841,177.671,23.371,153.545
C05133=1090.840,360.541,407.806,177.674,23.376,153.546
C05134=1090.846,360.789,407.770,177.677,23.381,153.547
C05135=1090.851,361.036,407.735,177.680,23.386,153.547
C05136=1090.857,361.284,407.699,177.684,23.391,153.548
C05137=1090.863,361.531,407.663,177.686,23.396,153.549
C05138=1090.869,361.778,407.628,177.689,23.401,153.550
C05139=1090.875,362.026,407.592,177.693,23.407,153.551
C05140=1090.880,362.273,407.557,177.696,23.412,153.551
C05141=1090.887,362.520,407.522,177.698,23.417,153.552
C05142=1090.893,362.768,407.486,177.702,23.422,153.553
C05143=1090.899,363.014,407.450,177.705,23.427,153.554
C05144=1090.905,363.262,407.414,177.707,23.432,153.554
C05145=1090.911,363.510,407.379,177.711,23.437,153.555
C05146=1090.917,363.757,407.343,177.714,23.443,153.556
C05147=1090.922,364.004,407.307,177.717,23.448,153.557
C05148=1090.928,364.252,407.272,177.720,23.453,153.558
C05149=1090.935,364.499,407.235,177.723,23.458,153.558
C05150=1090.940,364.746,407.200,177.726,23.464,153.559
C05151=1090.946,364.994,407.164,177.729,23.469,153.560
C05152=1090.952,365.241,407.128,177.732,23.473,153.561
C05153=1090.958,365.488,407.092,177.735,23.479,153.562
C05154=1090.964,365.735,407.057,177.739,23.484,153.562
C05155=1090.970,365.983,407.021,177.741,23.489,153.563
C05156=1090.975,366.230,406.984,177.744,23.495,153.564
C05157=1090.981,366.477,406.949,177.748,23.500,153.565
C05158=1090.987,366.725,406.913,177.751,23.506,153.566
C05159=1090.993,366.972,406.876,177.754,23.511,153.567
C05160=1090.999,367.219,406.841,177.756,23.517,153.568
C05161=1091.004,367.466,406.804,177.760,23.522,153.569
C05162=1091.010,367.714,406.768,177.763,23.527,153.569
C05163=1091.016,367.962,406.733,177.766,23.533,153.570
C05164=1091.022,368.208,406.696,177.769,23.538,153.571
C05165=1091.028,368.456,406.661,177.772,23.543,153.572
C05166=1091.034,368.703,406.624,177.775,23.549,153.573
C05167=1091.040,368.951,406.588,177.778,23.555,153.574
C05168=1091.045,369.197,406.552,177.781,23.560,153.575
C05169=1091.052,369.444,406.515,177.784,23.566,153.576
C05170=1091.057,369.692,406.479,177.787,23.571,153.576
C05171=1091.067,370.097,406.419,177.792,23.580,153.578
C05172=1091.077,370.502,406.360,177.797,23.589,153.579
C05173=1091.086,370.908,406.301,177.802,23.598,153.581
C05174=1091.096,371.312,406.241,177.807,23.607,153.582
C05175=1091.103,371.559,406.204,177.811,23.613,153.583
C05176=1091.108,371.807,406.169,177.813,23.618,153.584
C05177=1091.114,372.054,406.132,177.816,23.624,153.585
C05178=1091.120,372.301,406.096,177.819,23.630,153.586
C05179=1091.126,372.548,406.059,177.822,23.635,153.587
C05180=1091.132,372.796,406.023,177.826,23.641,153.588
C05181=1091.138,373.043,405.986,177.829,23.646,153.589
C05182=1091.144,373.290,405.949,177.832,23.652,153.590
C05183=1091.150,373.537,405.913,177.834,23.658,153.591
C05184=1091.156,373.784,405.876,177.838,23.663,153.591
C05185=1091.162,374.032,405.839,177.841,23.669,153.592
C05186=1091.168,374.279,405.803,177.844,23.675,153.593
C05187=1091.174,374.526,405.766,177.847,23.681,153.594
C05188=1091.180,374.772,405.730,177.850,23.687,153.595
C05189=1091.185,375.020,405.693,177.853,23.693,153.596
C05190=1091.192,375.267,405.656,177.856,23.698,153.597
C05191=1091.197,375.514,405.619,177.859,23.704,153.598
C05192=1091.203,375.762,405.582,177.862,23.710,153.599
C05193=1091.209,376.009,405.546,177.865,23.716,153.600
C05194=1091.215,376.256,405.509,177.868,23.721,153.601
C05195=1091.221,376.503,405.472,177.871,23.728,153.602
C05196=1091.227,376.750,405.435,177.874,23.734,153.603
C05197=1091.232,376.998,405.398,177.877,23.739,153.604
C05198=1091.239,377.244,405.361,177.880,23.745,153.605
C05199=1091.245,377.492,405.324,177.883,23.751,153.606
C05200=1091.251,377.739,405.288,177.886,23.758,153.607
C05201=1091.256,377.986,405.251,177.890,23.763,153.608
C05202=1091.262,378.233,405.214,177.893,23.769,153.609
C05203=1091.269,378.480,405.176,177.895,23.775,153.610
C05204=1091.274,378.727,405.139,177.898,23.781,153.611
C05205=1091.280,378.974,405.102,177.901,23.787,153.612
C05206=1091.287,379.221,405.065,177.904,23.793,153.613
C05207=1091.292,379.468,405.028,177.907,23.799,153.614
C05208=1091.298,379.716,404.991,177.910,23.805,153.615
C05209=1091.304,379.962,404.954,177.913,23.811,153.616
C05210=1091.310,380.209,404.917,177.916,23.817,153.617
C05211=1091.316,380.456,404.879,177.919,23.824,153.619
C05212=1091.321,380.704,404.842,177.923,23.830,153.620
C05213=1091.328,380.951,404.805,177.926,23.836,153.621
C05214=1091.334,381.198,404.768,177.929,23.842,153.622
C05215=1091.340,381.445,404.730,177.932,23.848,153.623
C05216=1091.347,381.692,404.693,177.935,23.854,153.624
C05217=1091.352,381.939,404.656,177.938,23.861,153.625
C05218=1091.358,382.186,404.619,177.941,23.867,153.626
C05219=1091.364,382.433,404.581,177.944,23.873,153.627
C05220=1091.371,382.680,404.544,177.947,23.879,153.628
C05221=1091.377,382.927,404.506,177.950,23.885,153.629
C05222=1091.382,383.175,404.469,177.953,23.892,153.630
C05223=1091.388,383.390,404.436,177.955,23.897,153.631
C05224=1091.393,383.607,404.403,177.958,23.903,153.632
C05225=1091.398,383.823,404.370,177.961,23.908,153.633
C05226=1091.403,384.039,404.338,177.964,23.914,153.634
C05227=1091.408,384.256,404.305,177.966,23.920,153.635
C05228=1091.413,384.472,404.271,177.969,23.925,153.636
C05229=1091.418,384.689,404.238,177.972,23.931,153.637
C05230=1091.424,384.905,404.205,177.974,23.936,153.638
C05231=1091.429,385.152,404.168,177.977,23.943,153.639
C05232=1091.435,385.399,404.130,177.981,23.950,153.641
C05233=1091.442,385.646,404.092,177.984,23.956,153.642
C05234=1091.448,385.893,404.054,177.987,23.963,153.643
C05235=1091.453,386.140,404.017,177.990,23.969,153.644
C05236=1091.459,386.387,403.979,177.992,23.976,153.645
C05237=1091.465,386.633,403.941,177.995,23.982,153.646
C05238=1091.471,386.881,403.904,177.998,23.989,153.648
C05239=1091.477,387.128,403.866,178.001,23.995,153.649
C05240=1091.483,387.375,403.828,178.004,24.002,153.650
C05241=1091.489,387.622,403.790,178.007,24.008,153.651
C05242=1091.496,387.869,403.752,178.010,24.015,153.652
C05243=1091.502,388.116,403.715,178.014,24.022,153.654
C05244=1091.507,388.362,403.677,178.017,24.028,153.655
C05245=1091.514,388.609,403.638,178.020,24.035,153.656
C05246=1091.520,388.856,403.600,178.023,24.042,153.657
C05247=1091.526,389.103,403.562,178.026,24.048,153.658
C05248=1091.531,389.350,403.524,178.028,24.055,153.660
C05249=1091.538,389.597,403.486,178.032,24.061,153.661
C05250=1091.544,389.844,403.448,178.034,24.068,153.662
C05251=1091.550,390.091,403.410,178.038,24.075,153.663
C05252=1091.556,390.338,403.372,178.041,24.082,153.664
C05253=1091.562,390.584,403.334,178.044,24.089,153.666
C05254=1091.569,390.832,403.296,178.047,24.096,153.667
C05255=1091.574,391.079,403.257,178.050,24.102,153.668
C05256=1091.580,391.325,403.219,178.053,24.109,153.669
C05257=1091.587,391.572,403.181,178.056,24.117,153.671
C05258=1091.593,391.819,403.143,178.059,24.123,153.672
C05259=1091.599,392.067,403.105,178.062,24.130,153.673
C05260=1091.605,392.313,403.066,178.065,24.137,153.674
C05261=1091.611,392.560,403.028,178.068,24.144,153.676
C05262=1091.617,392.807,402.989,178.071,24.151,153.677
C05263=1091.622,393.054,402.951,178.074,24.158,153.678
C05264=1091.629,393.301,402.913,178.077,24.165,153.680
C05265=1091.635,393.547,402.874,178.080,24.172,153.681
C05266=1091.641,393.795,402.836,178.083,24.179,153.682
C05267=1091.647,394.041,402.797,178.086,24.186,153.684
C05268=1091.654,394.289,402.759,178.089,24.194,153.685
C05269=1091.659,394.535,402.720,178.092,24.200,153.686
C05270=1091.666,394.782,402.682,178.095,24.207,153.688
C05271=1091.671,395.029,402.643,178.098,24.215,153.689
C05272=1091.678,395.276,402.604,178.101,24.222,153.690
C05273=1091.683,395.523,402.566,178.104,24.229,153.692
C05274=1091.690,395.770,402.527,178.107,24.236,153.693
C05275=1091.695,396.017,402.488,178.110,24.244,153.694
C05276=1091.702,396.263,402.450,178.113,24.251,153.696
C05277=1091.707,396.510,402.410,178.116,24.258,153.697
C05278=1091.714,396.757,402.372,178.119,24.266,153.698
C05279=1091.720,396.980,402.337,178.122,24.272,153.700
C05280=1091.725,397.203,402.302,178.125,24.279,153.701
C05281=1091.730,397.426,402.267,178.127,24.285,153.702
C05282=1091.736,397.649,402.232,178.130,24.292,153.703
C05283=1091.741,397.872,402.197,178.133,24.299,153.705
C05284=1091.747,398.095,402.162,178.136,24.306,153.706
C05285=1091.752,398.318,402.126,178.138,24.312,153.707
C05286=1091.758,398.541,402.091,178.141,24.319,153.709
C05287=1091.763,398.787,402.052,178.144,24.327,153.710
C05288=1091.770,399.034,402.013,178.147,24.334,153.711
C05289=1091.776,399.282,401.974,178.150,24.341,153.713
C05290=1091.781,399.528,401.935,178.153,24.349,153.714
C05291=1091.788,399.775,401.896,178.156,24.357,153.716
C05292=1091.794,400.022,401.857,178.159,24.364,153.717
C05293=1091.800,400.269,401.818,178.162,24.372,153.719
C05294=1091.807,400.515,401.779,178.165,24.379,153.720
C05295=1091.813,400.762,401.739,178.168,24.387,153.722
C05296=1091.818,401.009,401.700,178.171,24.395,153.723
C05297=1091.824,401.256,401.661,178.174,24.402,153.725
C05298=1091.830,401.503,401.621,178.176,24.410,153.726
C05299=1091.837,401.749,401.582,178.180,24.418,153.728
C05300=1091.843,401.996,401.543,178.183,24.426,153.729
C05301=1091.849,402.243,401.503,178.186,24.434,153.731
C05302=1091.855,402.490,401.464,178.189,24.442,153.732
C05303=1091.861,402.737,401.425,178.191,24.449,153.734
C05304=1091.867,402.983,401.386,178.195,24.457,153.735
C05305=1091.874,403.230,401.346,178.198,24.465,153.737
C05306=1091.880,403.477,401.307,178.201,24.473,153.738
C05307=1091.886,403.724,401.267,178.204,24.481,153.740
C05308=1091.892,403.971,401.228,178.207,24.489,153.741
C05309=1091.898,404.217,401.188,178.210,24.497,153.743
C05310=1091.904,404.464,401.148,178.212,24.505,153.745
C05311=1091.910,404.711,401.109,178.216,24.513,153.746
C05312=1091.916,404.958,401.069,178.219,24.521,153.748
C05313=1091.922,405.205,401.029,178.222,24.529,153.749
C05314=1091.929,405.452,400.989,178.225,24.537,153.751
C05315=1091.934,405.698,400.950,178.228,24.545,153.752
C05316=1091.941,405.944,400.910,178.231,24.553,153.754
C05317=1091.947,406.192,400.871,178.234,24.562,153.756
C05318=1091.953,406.438,400.830,178.237,24.570,153.757
C05319=1091.959,406.685,400.791,178.240,24.578,153.759
C05320=1091.965,406.932,400.751,178.243,24.586,153.760
C05321=1091.972,407.179,400.711,178.246,24.595,153.762
C05322=1091.978,407.425,400.671,178.249,24.603,153.764
C05323=1091.983,407.672,400.632,178.252,24.611,153.765
C05324=1091.990,407.918,400.592,178.256,24.620,153.767
C05325=1091.996,408.165,400.552,178.258,24.628,153.769
C05326=1092.001,408.412,400.512,178.261,24.637,153.770
C05327=1092.008,408.659,400.472,178.264,24.645,153.772
C05328=1092.014,408.905,400.432,178.267,24.654,153.774
C05329=1092.021,409.152,400.392,178.271,24.663,153.776
C05330=1092.026,409.399,400.351,178.273,24.671,153.777
C05331=1092.032,409.646,400.311,178.277,24.679,153.779
C05332=1092.039,409.892,400.271,178.279,24.688,153.781
C05333=1092.045,410.139,400.231,178.282,24.697,153.782
C05334=1092.051,410.386,400.190,178.286,24.706,153.784
C05335=1092.056,410.610,400.154,178.288,24.713,153.786
C05336=1092.062,410.832,400.118,178.291,24.721,153.787
C05337=1092.068,411.056,400.081,178.294,24.729,153.789
C05338=1092.073,411.280,400.045,178.296,24.737,153.790
C05339=1092.079,411.502,400.009,178.299,24.745,153.792
C05340=1092.085,411.726,399.972,178.303,24.753,153.794
C05341=1092.090,411.949,399.936,178.305,24.761,153.795
C05342=1092.096,412.173,399.899,178.308,24.769,153.797
C05343=1092.102,412.420,399.858,178.311,24.778,153.799
C05344=1092.108,412.666,399.818,178.314,24.786,153.800
C05345=1092.115,412.913,399.778,178.317,24.795,153.802
C05346=1092.120,413.159,399.737,178.320,24.804,153.804
C05347=1092.127,413.405,399.696,178.323,24.813,153.806
C05348=1092.133,413.652,399.656,178.326,24.822,153.808
C05349=1092.139,413.899,399.615,178.329,24.831,153.810
C05350=1092.145,414.145,399.575,178.333,24.840,153.811
C05351=1092.152,414.393,399.534,178.335,24.849,153.813
C05352=1092.158,414.639,399.493,178.338,24.858,153.815
C05353=1092.165,414.885,399.453,178.341,24.868,153.817
C05354=1092.170,415.132,399.412,178.345,24.877,153.819
C05355=1092.177,415.378,399.372,178.348,24.886,153.821
C05356=1092.183,415.625,399.330,178.350,24.895,153.823
C05357=1092.190,415.872,399.290,178.354,24.904,153.824
C05358=1092.196,416.118,399.249,178.357,24.914,153.826
C05359=1092.202,416.365,399.209,178.360,24.923,153.828
C05360=1092.208,416.611,399.167,178.363,24.932,153.830
C05361=1092.215,416.858,399.127,178.367,24.942,153.832
C05362=1092.220,417.105,399.086,178.369,24.951,153.834
C05363=1092.226,417.351,399.045,178.372,24.960,153.836
C05364=1092.233,417.597,399.004,178.375,24.970,153.838
C05365=1092.239,417.845,398.963,178.379,24.979,153.840
C05366=1092.246,418.090,398.922,178.382,24.989,153.842
C05367=1092.252,418.337,398.881,178.385,24.999,153.844
C05368=1092.258,418.583,398.839,178.388,25.008,153.846
C05369=1092.264,418.830,398.798,178.391,25.018,153.848
C05370=1092.271,419.077,398.758,178.395,25.027,153.850
C05371=1092.276,419.323,398.716,178.398,25.038,153.852
C05372=1092.282,419.569,398.675,178.401,25.047,153.854
C05373=1092.290,419.816,398.633,178.403,25.056,153.856
C05374=1092.295,420.063,398.593,178.406,25.066,153.858
C05375=1092.301,420.309,398.551,178.409,25.076,153.860
C05376=1092.308,420.556,398.509,178.412,25.086,153.862
C05377=1092.315,420.802,398.468,178.416,25.096,153.864
C05378=1092.321,421.048,398.427,178.419,25.106,153.866
C05379=1092.327,421.295,398.385,178.422,25.116,153.868
C05380=1092.333,421.541,398.344,178.425,25.126,153.870
C05381=1092.340,421.788,398.303,178.428,25.135,153.872
C05382=1092.346,422.034,398.261,178.431,25.145,153.874
C05383=1092.352,422.280,398.220,178.434,25.156,153.877
C05384=1092.359,422.527,398.178,178.437,25.166,153.879
C05385=1092.365,422.773,398.136,178.440,25.176,153.881
C05386=1092.371,423.020,398.095,178.444,25.186,153.883
C05387=1092.377,423.266,398.053,178.448,25.196,153.885
C05388=1092.383,423.512,398.012,178.451,25.207,153.887
C05389=1092.390,423.759,397.970,178.454,25.217,153.890
C05390=1092.396,424.006,397.928,178.457,25.227,153.892
C05391=1092.404,424.301,397.878,178.460,25.240,153.894
C05392=1092.411,424.596,397.829,178.464,25.252,153.897
C05393=1092.419,424.891,397.778,178.468,25.265,153.900
C05394=1092.426,425.186,397.728,178.471,25.277,153.902
C05395=1092.433,425.431,397.686,178.474,25.287,153.904
C05396=1092.439,425.678,397.644,178.477,25.298,153.907
C05397=1092.445,425.925,397.603,178.481,25.309,153.909
C05398=1092.452,426.171,397.560,178.484,25.320,153.911
C05399=1092.458,426.417,397.519,178.487,25.330,153.913
C05400=1092.465,426.663,397.476,178.490,25.341,153.916
C05401=1092.471,426.910,397.434,178.493,25.351,153.918
C05402=1092.477,427.156,397.392,178.496,25.362,153.920
C05403=1092.483,427.403,397.350,178.500,25.373,153.923
C05404=1092.490,427.649,397.308,178.503,25.384,153.925
C05405=1092.496,427.896,397.266,178.506,25.395,153.927
C05406=1092.503,428.142,397.223,178.509,25.406,153.930
C05407=1092.509,428.387,397.181,178.513,25.416,153.932
C05408=1092.516,428.634,397.139,178.516,25.427,153.934
C05409=1092.522,428.880,397.097,178.519,25.438,153.937
C05410=1092.528,429.127,397.054,178.522,25.449,153.939
C05411=1092.535,429.373,397.011,178.526,25.461,153.941
C05412=1092.541,429.619,396.970,178.528,25.472,153.944
C05413=1092.548,429.865,396.927,178.531,25.483,153.946
C05414=1092.554,430.112,396.884,178.534,25.494,153.949
C05415=1092.560,430.357,396.842,178.538,25.505,153.951
C05416=1092.567,430.604,396.800,178.541,25.517,153.954
C05417=1092.573,430.850,396.756,178.544,25.528,153.956
C05418=1092.580,431.096,396.714,178.548,25.540,153.958
C05419=1092.586,431.342,396.672,178.551,25.551,153.961
C05420=1092.593,431.589,396.629,178.553,25.562,153.963
C05421=1092.599,431.834,396.586,178.557,25.574,153.966
C05422=1092.605,432.081,396.543,178.560,25.585,153.968
C05423=1092.612,432.327,396.501,178.563,25.597,153.971
C05424=1092.619,432.574,396.458,178.567,25.608,153.973
C05425=1092.624,432.819,396.415,178.569,25.620,153.976
C05426=1092.631,433.066,396.373,178.573,25.632,153.979
C05427=1092.637,433.312,396.330,178.576,25.643,153.981
C05428=1092.644,433.558,396.286,178.579,25.655,153.984
C05429=1092.650,433.804,396.244,178.582,25.667,153.986
C05430=1092.657,434.050,396.201,178.585,25.679,153.989
C05431=1092.663,434.297,396.158,178.589,25.691,153.991
C05432=1092.670,434.542,396.115,178.592,25.703,153.994
C05433=1092.675,434.788,396.072,178.595,25.715,153.997
C05434=1092.682,435.035,396.029,178.598,25.727,153.999
C05435=1092.689,435.281,395.986,178.602,25.739,154.002
C05436=1092.695,435.527,395.942,178.605,25.751,154.005
C05437=1092.702,435.773,395.899,178.608,25.763,154.007
C05438=1092.708,436.019,395.856,178.611,25.775,154.010
C05439=1092.719,436.431,395.784,178.616,25.796,154.015
C05440=1092.729,436.843,395.711,178.622,25.817,154.019
C05441=1092.740,437.256,395.638,178.627,25.837,154.024
C05442=1092.752,437.668,395.565,178.633,25.858,154.028
C05443=1092.757,437.876,395.529,178.636,25.869,154.031
C05444=1092.768,438.293,395.455,178.641,25.890,154.036
C05445=1092.773,438.501,395.418,178.643,25.901,154.038
C05446=1092.779,438.710,395.382,178.646,25.912,154.040
C05447=1092.785,438.918,395.344,178.649,25.922,154.043
C05448=1092.790,439.127,395.307,178.652,25.933,154.045
C05449=1092.796,439.335,395.271,178.655,25.944,154.047
C05450=1092.802,439.581,395.227,178.657,25.957,154.050
C05451=1092.809,439.827,395.183,178.661,25.970,154.053
C05452=1092.815,440.073,395.139,178.665,25.983,154.056
C05453=1092.822,440.320,395.095,178.667,25.995,154.059
C05454=1092.829,440.565,395.052,178.671,26.009,154.062
C05455=1092.836,440.811,395.008,178.674,26.022,154.065
C05456=1092.842,441.057,394.964,178.677,26.035,154.068
C05457=1092.849,441.303,394.920,178.680,26.048,154.071
